C09134=1206.719,382.178,-78.740,-175.897,8.142,148.400
C09135=1206.716,382.425,-78.774,-175.896,8.145,148.400
C09136=1206.711,382.673,-78.809,-175.895,8.148,148.401
C09137=1206.707,382.920,-78.843,-175.894,8.151,148.401
C09138=1206.703,383.168,-78.877,-175.893,8.153,148.402
C09139=1206.700,383.415,-78.911,-175.892,8.156,148.402
C09140=1206.695,383.663,-78.946,-175.891,8.159,148.403
C09141=1206.691,383.911,-78.979,-175.890,8.162,148.403
C09142=1206.687,384.158,-79.014,-175.889,8.165,148.404
C09143=1206.684,384.406,-79.048,-175.888,8.168,148.404
C09144=1206.679,384.654,-79.082,-175.887,8.170,148.405
C09145=1206.675,384.901,-79.117,-175.887,8.173,148.405
C09146=1206.671,385.149,-79.151,-175.886,8.176,148.406
C09147=1206.667,385.396,-79.186,-175.885,8.179,148.406
C09148=1206.663,385.643,-79.219,-175.884,8.181,148.407
C09149=1206.659,385.892,-79.254,-175.883,8.185,148.407
C09150=1206.654,386.139,-79.289,-175.882,8.187,148.408
C09151=1206.651,386.387,-79.323,-175.882,8.190,148.408
C09152=1206.647,386.634,-79.357,-175.881,8.193,148.409
C09153=1206.643,386.881,-79.391,-175.880,8.196,148.409
C09154=1206.639,387.129,-79.426,-175.879,8.198,148.410
C09155=1206.634,387.377,-79.461,-175.878,8.201,148.410
C09156=1206.631,387.625,-79.495,-175.877,8.204,148.411
C09157=1206.626,387.872,-79.529,-175.876,8.207,148.411
C09158=1206.623,388.119,-79.563,-175.876,8.209,148.412
C09159=1206.619,388.367,-79.598,-175.875,8.212,148.412
C09160=1206.614,388.615,-79.633,-175.874,8.215,148.413
C09161=1206.611,388.863,-79.667,-175.874,8.217,148.413
C09162=1206.606,389.110,-79.701,-175.873,8.220,148.414
C09163=1206.602,389.358,-79.736,-175.872,8.223,148.414
C09164=1206.598,389.605,-79.770,-175.872,8.225,148.415
C09165=1206.594,389.853,-79.804,-175.870,8.228,148.415
C09166=1206.590,390.101,-79.839,-175.870,8.231,148.416
C09167=1206.586,390.348,-79.873,-175.869,8.233,148.416
C09168=1206.582,390.596,-79.908,-175.868,8.236,148.417
C09169=1206.577,390.843,-79.942,-175.867,8.239,148.417
C09170=1206.574,391.091,-79.977,-175.867,8.242,148.418
C09171=1206.570,391.338,-80.012,-175.866,8.244,148.418
C09172=1206.566,391.586,-80.047,-175.866,8.247,148.419
C09173=1206.562,391.833,-80.081,-175.865,8.250,148.419
C09174=1206.558,392.081,-80.115,-175.864,8.252,148.420
C09175=1206.553,392.364,-80.154,-175.864,8.255,148.420
C09176=1206.549,392.646,-80.194,-175.863,8.258,148.421
C09177=1206.544,392.928,-80.234,-175.862,8.261,148.421
C09178=1206.540,393.211,-80.273,-175.861,8.264,148.422
C09179=1206.535,393.459,-80.307,-175.861,8.267,148.423
C09180=1206.531,393.707,-80.342,-175.860,8.269,148.423
C09181=1206.527,393.954,-80.377,-175.859,8.272,148.423
C09182=1206.524,394.201,-80.412,-175.859,8.275,148.424
C09183=1206.519,394.449,-80.446,-175.858,8.277,148.424
C09184=1206.515,394.697,-80.481,-175.858,8.280,148.425
C09185=1206.511,394.944,-80.515,-175.857,8.283,148.425
C09186=1206.508,395.192,-80.550,-175.857,8.285,148.426
C09187=1206.503,395.439,-80.585,-175.856,8.287,148.426
C09188=1206.499,395.687,-80.620,-175.855,8.290,148.427
C09189=1206.495,395.935,-80.654,-175.855,8.292,148.427
C09190=1206.492,396.182,-80.689,-175.854,8.296,148.428
C09191=1206.487,396.429,-80.723,-175.853,8.297,148.428
C09192=1206.483,396.677,-80.758,-175.853,8.301,148.429
C09193=1206.479,396.925,-80.793,-175.853,8.303,148.430
C09194=1206.475,397.172,-80.828,-175.852,8.305,148.430
C09195=1206.471,397.419,-80.862,-175.851,8.308,148.430
C09196=1206.467,397.667,-80.897,-175.851,8.310,148.431
C09197=1206.463,397.915,-80.931,-175.851,8.312,148.432
C09198=1206.459,398.162,-80.967,-175.849,8.315,148.432
C09199=1206.454,398.410,-81.001,-175.849,8.318,148.432
C09200=1206.450,398.658,-81.036,-175.848,8.321,148.433
C09201=1206.447,398.904,-81.071,-175.848,8.323,148.434
C09202=1206.443,399.153,-81.106,-175.848,8.325,148.434
C09203=1206.438,399.400,-81.140,-175.847,8.328,148.435
C09204=1206.435,399.647,-81.176,-175.847,8.330,148.435
C09205=1206.430,399.895,-81.210,-175.846,8.333,148.436
C09206=1206.427,400.143,-81.244,-175.846,8.335,148.436
C09207=1206.423,400.389,-81.280,-175.845,8.338,148.437
C09208=1206.419,400.638,-81.314,-175.845,8.340,148.437
C09209=1206.414,400.885,-81.349,-175.845,8.342,148.438
C09210=1206.410,401.133,-81.384,-175.844,8.345,148.438
C09211=1206.406,401.380,-81.419,-175.843,8.347,148.439
C09212=1206.402,401.628,-81.454,-175.843,8.350,148.439
C09213=1206.399,401.875,-81.489,-175.843,8.352,148.440
C09214=1206.394,402.123,-81.523,-175.842,8.355,148.440
C09215=1206.391,402.370,-81.559,-175.841,8.357,148.441
C09216=1206.386,402.618,-81.593,-175.841,8.359,148.441
C09217=1206.382,402.866,-81.628,-175.841,8.361,148.442
C09218=1206.378,403.112,-81.663,-175.840,8.364,148.442
C09219=1206.374,403.361,-81.698,-175.839,8.366,148.443
C09220=1206.370,403.608,-81.734,-175.839,8.369,148.443
C09221=1206.366,403.856,-81.768,-175.839,8.371,148.444
C09222=1206.363,404.103,-81.802,-175.839,8.373,148.444
C09223=1206.358,404.350,-81.837,-175.838,8.376,148.445
C09224=1206.354,404.598,-81.872,-175.837,8.378,148.445
C09225=1206.350,404.845,-81.907,-175.837,8.381,148.446
C09226=1206.346,405.093,-81.942,-175.837,8.383,148.446
C09227=1206.342,405.341,-81.978,-175.837,8.385,148.447
C09228=1206.338,405.588,-82.012,-175.836,8.387,148.447
C09229=1206.334,405.836,-82.048,-175.836,8.389,148.447
C09230=1206.330,406.083,-82.082,-175.835,8.392,148.448
C09231=1206.326,406.331,-82.118,-175.835,8.395,148.449
C09232=1206.321,406.578,-82.152,-175.834,8.397,148.449
C09233=1206.318,406.825,-82.188,-175.834,8.399,148.449
C09234=1206.314,407.073,-82.222,-175.834,8.401,148.450
C09235=1206.310,407.320,-82.257,-175.833,8.404,148.451
C09236=1206.306,407.568,-82.292,-175.833,8.406,148.451
C09237=1206.302,407.815,-82.327,-175.833,8.408,148.451
C09238=1206.298,408.063,-82.362,-175.832,8.410,148.452
C09239=1206.294,408.311,-82.398,-175.832,8.413,148.453
C09240=1206.290,408.558,-82.432,-175.831,8.415,148.453
C09241=1206.286,408.806,-82.468,-175.831,8.417,148.453
C09242=1206.282,409.053,-82.502,-175.830,8.420,148.454
C09243=1206.278,409.300,-82.538,-175.830,8.422,148.454
C09244=1206.274,409.549,-82.573,-175.830,8.424,148.455
C09245=1206.270,409.795,-82.608,-175.829,8.426,148.455
C09246=1206.266,410.043,-82.643,-175.829,8.428,148.456
C09247=1206.262,410.291,-82.678,-175.829,8.431,148.456
C09248=1206.258,410.538,-82.713,-175.828,8.433,148.457
C09249=1206.254,410.786,-82.748,-175.828,8.435,148.457
C09250=1206.250,411.033,-82.783,-175.828,8.437,148.458
C09251=1206.246,411.281,-82.818,-175.828,8.439,148.458
C09252=1206.242,411.528,-82.854,-175.827,8.441,148.459
C09253=1206.238,411.775,-82.889,-175.827,8.444,148.459
C09254=1206.234,412.023,-82.924,-175.826,8.446,148.460
C09255=1206.230,412.271,-82.959,-175.826,8.448,148.460
C09256=1206.226,412.518,-82.994,-175.826,8.450,148.461
C09257=1206.222,412.766,-83.029,-175.825,8.452,148.461
C09258=1206.218,413.013,-83.065,-175.825,8.455,148.462
C09259=1206.214,413.261,-83.099,-175.824,8.457,148.462
C09260=1206.210,413.508,-83.135,-175.824,8.459,148.463
C09261=1206.206,413.755,-83.170,-175.824,8.461,148.463
C09262=1206.202,414.003,-83.205,-175.823,8.463,148.463
C09263=1206.198,414.250,-83.240,-175.823,8.465,148.464
C09264=1206.194,414.497,-83.276,-175.823,8.468,148.464
C09265=1206.190,414.745,-83.310,-175.822,8.470,148.465
C09266=1206.186,414.993,-83.346,-175.822,8.472,148.465
C09267=1206.182,415.240,-83.381,-175.822,8.474,148.466
C09268=1206.178,415.488,-83.416,-175.821,8.476,148.466
C09269=1206.174,415.735,-83.452,-175.821,8.478,148.467
C09270=1206.170,415.982,-83.487,-175.821,8.480,148.467
C09271=1206.165,416.261,-83.526,-175.820,8.483,148.468
C09272=1206.162,416.540,-83.566,-175.820,8.485,148.468
C09273=1206.160,416.817,-83.606,-175.820,8.487,148.469
C09274=1206.162,417.095,-83.644,-175.819,8.490,148.469
C09275=1205.741,417.096,-83.682,-175.823,8.500,148.473
C09276=1205.738,416.816,-83.643,-175.823,8.498,148.472
C09277=1205.740,416.534,-83.602,-175.823,8.496,148.472
C09278=1205.743,416.253,-83.563,-175.824,8.494,148.471
C09279=1205.748,415.972,-83.522,-175.825,8.491,148.471
C09280=1205.752,415.724,-83.488,-175.825,8.488,148.470
C09281=1205.756,415.477,-83.452,-175.824,8.487,148.470
C09282=1205.760,415.230,-83.417,-175.825,8.485,148.470
C09283=1205.764,414.981,-83.382,-175.825,8.483,148.469
C09284=1205.768,414.735,-83.347,-175.826,8.480,148.468
C09285=1205.772,414.487,-83.311,-175.826,8.478,148.468
C09286=1205.776,414.240,-83.277,-175.826,8.476,148.468
C09287=1205.780,413.992,-83.241,-175.827,8.474,148.467
C09288=1205.784,413.744,-83.205,-175.827,8.472,148.467
C09289=1205.789,413.497,-83.171,-175.828,8.470,148.466
C09290=1205.793,413.250,-83.135,-175.828,8.467,148.466
C09291=1205.796,413.002,-83.100,-175.828,8.465,148.465
C09292=1205.801,412.755,-83.065,-175.829,8.463,148.465
C09293=1205.804,412.507,-83.030,-175.829,8.461,148.464
C09294=1205.808,412.260,-82.994,-175.829,8.459,148.464
C09295=1205.813,412.012,-82.960,-175.829,8.456,148.463
C09296=1205.816,411.765,-82.924,-175.830,8.454,148.463
C09297=1205.820,411.517,-82.889,-175.830,8.452,148.462
C09298=1205.825,411.270,-82.854,-175.830,8.450,148.462
C09299=1205.828,411.022,-82.818,-175.831,8.448,148.461
C09300=1205.833,410.775,-82.784,-175.831,8.446,148.461
C09301=1205.836,410.527,-82.748,-175.832,8.443,148.460
C09302=1205.840,410.279,-82.714,-175.832,8.441,148.460
C09303=1205.845,410.032,-82.678,-175.832,8.439,148.459
C09304=1205.848,409.785,-82.643,-175.833,8.437,148.459
C09305=1205.852,409.537,-82.608,-175.833,8.435,148.459
C09306=1205.857,409.290,-82.573,-175.833,8.432,148.458
C09307=1205.861,409.042,-82.538,-175.833,8.430,148.457
C09308=1205.864,408.795,-82.503,-175.834,8.428,148.457
C09309=1205.868,408.547,-82.469,-175.834,8.426,148.457
C09310=1205.872,408.300,-82.433,-175.834,8.424,148.456
C09311=1205.876,408.052,-82.399,-175.835,8.421,148.456
C09312=1205.880,407.805,-82.363,-175.835,8.419,148.455
C09313=1205.884,407.558,-82.328,-175.836,8.416,148.455
C09314=1205.888,407.310,-82.293,-175.836,8.414,148.454
C09315=1205.892,407.062,-82.257,-175.836,8.412,148.454
C09316=1205.896,406.815,-82.223,-175.837,8.410,148.453
C09317=1205.900,406.568,-82.187,-175.837,8.407,148.453
C09318=1205.905,406.320,-82.153,-175.838,8.405,148.452
C09319=1205.908,406.073,-82.117,-175.838,8.403,148.452
C09320=1205.912,405.824,-82.083,-175.838,8.401,148.451
C09321=1205.916,405.578,-82.047,-175.839,8.398,148.451
C09322=1205.920,405.330,-82.013,-175.839,8.396,148.450
C09323=1205.925,405.082,-81.978,-175.840,8.393,148.450
C09324=1205.929,404.835,-81.943,-175.840,8.391,148.449
C09325=1205.932,404.587,-81.908,-175.841,8.389,148.449
C09326=1205.936,404.340,-81.873,-175.841,8.387,148.448
C09327=1205.940,404.092,-81.838,-175.841,8.384,148.448
C09328=1205.944,403.845,-81.803,-175.842,8.381,148.447
C09329=1205.948,403.597,-81.768,-175.842,8.379,148.447
C09330=1205.953,403.350,-81.733,-175.843,8.377,148.446
C09331=1205.957,403.102,-81.698,-175.843,8.375,148.446
C09332=1205.960,402.855,-81.663,-175.843,8.373,148.445
C09333=1205.965,402.607,-81.628,-175.844,8.369,148.445
C09334=1205.969,402.359,-81.593,-175.845,8.368,148.444
C09335=1205.972,402.113,-81.559,-175.845,8.365,148.444
C09336=1205.976,401.864,-81.524,-175.845,8.363,148.443
C09337=1205.981,401.618,-81.489,-175.846,8.360,148.443
C09338=1205.985,401.369,-81.454,-175.846,8.358,148.442
C09339=1205.989,401.122,-81.420,-175.847,8.356,148.442
C09340=1205.993,400.875,-81.384,-175.847,8.353,148.441
C09341=1205.997,400.626,-81.349,-175.848,8.350,148.441
C09342=1206.001,400.379,-81.315,-175.848,8.348,148.440
C09343=1206.004,400.132,-81.280,-175.848,8.346,148.440
C09344=1206.009,399.884,-81.245,-175.849,8.343,148.439
C09345=1206.013,399.636,-81.210,-175.849,8.341,148.439
C09346=1206.017,399.390,-81.175,-175.850,8.338,148.438
C09347=1206.021,399.141,-81.140,-175.851,8.336,148.438
C09348=1206.026,398.894,-81.106,-175.851,8.333,148.437
C09349=1206.029,398.647,-81.071,-175.851,8.331,148.437
C09350=1206.033,398.399,-81.037,-175.852,8.328,148.436
C09351=1206.037,398.151,-81.002,-175.853,8.326,148.436
C09352=1206.041,397.904,-80.967,-175.853,8.324,148.435
C09353=1206.045,397.656,-80.932,-175.854,8.321,148.435
C09354=1206.049,397.409,-80.898,-175.854,8.318,148.434
C09355=1206.053,397.162,-80.862,-175.855,8.316,148.434
C09356=1206.057,396.914,-80.828,-175.855,8.313,148.433
C09357=1206.061,396.666,-80.793,-175.856,8.311,148.433
C09358=1206.066,396.419,-80.758,-175.856,8.308,148.432
C09359=1206.069,396.172,-80.724,-175.857,8.306,148.432
C09360=1206.073,395.924,-80.689,-175.857,8.304,148.431
C09361=1206.077,395.676,-80.654,-175.858,8.301,148.430
C09362=1206.082,395.429,-80.620,-175.858,8.298,148.430
C09363=1206.086,395.181,-80.584,-175.859,8.295,148.430
C09364=1206.089,394.934,-80.550,-175.860,8.293,148.429
C09365=1206.093,394.686,-80.516,-175.860,8.290,148.428
C09366=1206.098,394.438,-80.481,-175.861,8.288,148.428
C09367=1206.102,394.190,-80.446,-175.862,8.285,148.428
C09368=1206.105,393.944,-80.412,-175.862,8.283,148.427
C09369=1206.109,393.696,-80.377,-175.863,8.280,148.426
C09370=1206.114,393.448,-80.342,-175.863,8.278,148.426
C09371=1206.118,393.200,-80.308,-175.864,8.275,148.425
C09372=1206.122,392.918,-80.268,-175.865,8.271,148.425
C09373=1206.127,392.635,-80.229,-175.865,8.269,148.424
C09374=1206.132,392.353,-80.189,-175.866,8.266,148.424
C09375=1206.136,392.070,-80.150,-175.867,8.263,148.423
C09376=1206.140,391.823,-80.114,-175.868,8.260,148.423
C09377=1206.144,391.576,-80.081,-175.868,8.258,148.422
C09378=1206.148,391.327,-80.046,-175.869,8.255,148.422
C09379=1206.152,391.080,-80.011,-175.870,8.252,148.421
C09380=1206.156,390.833,-79.977,-175.870,8.250,148.421
C09381=1206.160,390.585,-79.943,-175.871,8.247,148.420
C09382=1206.165,390.337,-79.908,-175.871,8.244,148.420
C09383=1206.168,390.090,-79.874,-175.873,8.241,148.419
C09384=1206.172,389.842,-79.839,-175.873,8.238,148.419
C09385=1206.176,389.595,-79.804,-175.874,8.236,148.418
C09386=1206.180,389.348,-79.770,-175.875,8.233,148.418
C09387=1206.184,389.099,-79.735,-175.876,8.230,148.417
C09388=1206.189,388.852,-79.701,-175.876,8.228,148.417
C09389=1206.192,388.605,-79.667,-175.877,8.225,148.416
C09390=1206.196,388.357,-79.632,-175.878,8.222,148.416
C09391=1206.201,388.109,-79.598,-175.878,8.220,148.415
C09392=1206.204,387.862,-79.563,-175.879,8.217,148.415
C09393=1206.209,387.614,-79.529,-175.880,8.214,148.414
C09394=1206.213,387.366,-79.494,-175.881,8.211,148.414
C09395=1206.217,387.119,-79.460,-175.881,8.209,148.413
C09396=1206.221,386.872,-79.426,-175.883,8.206,148.413
C09397=1206.225,386.623,-79.391,-175.883,8.203,148.412
C09398=1206.229,386.376,-79.357,-175.884,8.200,148.412
C09399=1206.233,386.128,-79.322,-175.885,8.198,148.411
C09400=1206.237,385.881,-79.288,-175.885,8.195,148.411
C09401=1206.241,385.634,-79.254,-175.887,8.192,148.410
C09402=1206.245,385.386,-79.219,-175.887,8.189,148.410
C09403=1206.249,385.138,-79.185,-175.888,8.187,148.409
C09404=1206.253,384.890,-79.150,-175.889,8.184,148.409
C09405=1206.257,384.643,-79.116,-175.890,8.181,148.408
C09406=1206.262,384.395,-79.083,-175.891,8.178,148.408
C09407=1206.265,384.147,-79.048,-175.892,8.175,148.407
C09408=1206.270,383.900,-79.014,-175.893,8.172,148.407
C09409=1206.274,383.652,-78.979,-175.894,8.169,148.406
C09410=1206.277,383.405,-78.945,-175.894,8.167,148.406
C09411=1206.282,383.157,-78.911,-175.895,8.164,148.405
C09412=1206.285,382.909,-78.877,-175.896,8.161,148.405
C09413=1206.290,382.662,-78.842,-175.897,8.158,148.404
C09414=1206.294,382.415,-78.808,-175.899,8.155,148.404
C09415=1206.298,382.166,-78.774,-175.899,8.152,148.403
C09416=1206.302,381.919,-78.740,-175.901,8.149,148.403
C09417=1206.306,381.672,-78.706,-175.901,8.146,148.402
C09418=1206.309,381.424,-78.671,-175.903,8.143,148.402
C09419=1206.314,381.176,-78.637,-175.904,8.141,148.402
C09420=1206.318,380.929,-78.604,-175.905,8.137,148.401
C09421=1206.322,380.681,-78.569,-175.906,8.135,148.401
C09422=1206.326,380.433,-78.535,-175.906,8.132,148.400
C09423=1206.331,380.186,-78.501,-175.907,8.130,148.400
C09424=1206.334,379.938,-78.466,-175.908,8.127,148.399
C09425=1206.339,379.690,-78.433,-175.909,8.124,148.399
C09426=1206.342,379.443,-78.399,-175.910,8.121,148.398
C09427=1206.346,379.195,-78.364,-175.912,8.118,148.398
C09428=1206.350,378.948,-78.330,-175.912,8.115,148.397
C09429=1206.355,378.700,-78.296,-175.914,8.111,148.397
C09430=1206.359,378.453,-78.263,-175.915,8.108,148.397
C09431=1206.363,378.205,-78.228,-175.916,8.105,148.396
C09432=1206.367,377.957,-78.195,-175.917,8.103,148.396
C09433=1206.371,377.710,-78.161,-175.918,8.100,148.395
C09434=1206.375,377.462,-78.126,-175.920,8.097,148.395
C09435=1206.379,377.215,-78.092,-175.920,8.094,148.394
C09436=1206.384,376.966,-78.058,-175.922,8.091,148.394
C09437=1206.387,376.719,-78.024,-175.923,8.088,148.393
C09438=1206.392,376.471,-77.990,-175.924,8.085,148.393
C09439=1206.396,376.224,-77.956,-175.925,8.083,148.393
C09440=1206.399,375.976,-77.922,-175.926,8.079,148.392
C09441=1206.404,375.728,-77.888,-175.927,8.077,148.392
C09442=1206.407,375.481,-77.854,-175.929,8.073,148.391
C09443=1206.411,375.233,-77.821,-175.930,8.070,148.391
C09444=1206.416,374.985,-77.787,-175.931,8.067,148.390
C09445=1206.419,374.738,-77.753,-175.933,8.065,148.390
C09446=1206.424,374.490,-77.719,-175.933,8.062,148.389
C09447=1206.428,374.242,-77.685,-175.935,8.059,148.389
C09448=1206.432,373.995,-77.652,-175.936,8.055,148.389
C09449=1206.436,373.747,-77.617,-175.938,8.052,148.388
C09450=1206.440,373.500,-77.583,-175.939,8.049,148.388
C09451=1206.444,373.252,-77.550,-175.940,8.047,148.387
C09452=1206.449,373.004,-77.516,-175.941,8.044,148.387
C09453=1206.452,372.756,-77.482,-175.943,8.040,148.387
C09454=1206.456,372.509,-77.448,-175.944,8.037,148.386
C09455=1206.461,372.261,-77.414,-175.945,8.035,148.386
C09456=1206.465,372.014,-77.381,-175.947,8.032,148.385
C09457=1206.468,371.765,-77.347,-175.948,8.029,148.385
C09458=1206.472,371.518,-77.313,-175.950,8.025,148.385
C09459=1206.477,371.270,-77.279,-175.951,8.022,148.384
C09460=1206.481,371.022,-77.246,-175.952,8.020,148.384
C09461=1206.485,370.775,-77.212,-175.953,8.017,148.383
C09462=1206.489,370.527,-77.179,-175.955,8.013,148.383
C09463=1206.493,370.279,-77.144,-175.956,8.010,148.383
C09464=1206.497,370.032,-77.111,-175.957,8.008,148.382
C09465=1206.501,369.784,-77.078,-175.959,8.004,148.382
C09466=1206.505,369.537,-77.044,-175.960,8.001,148.381
C09467=1206.510,369.288,-77.010,-175.961,7.998,148.381
C09468=1206.513,369.041,-76.976,-175.963,7.996,148.381
C09469=1206.517,368.793,-76.943,-175.964,7.992,148.380
C09470=1206.522,368.546,-76.910,-175.966,7.989,148.380
C09471=1206.526,368.298,-76.875,-175.967,7.987,148.380
C09472=1206.530,368.050,-76.842,-175.969,7.983,148.379
C09473=1206.534,367.802,-76.809,-175.970,7.980,148.379
C09474=1206.538,367.555,-76.775,-175.971,7.977,148.378
C09475=1206.542,367.307,-76.742,-175.973,7.974,148.378
C09476=1206.547,367.026,-76.703,-175.975,7.970,148.377
C09477=1206.551,366.746,-76.666,-175.977,7.967,148.377
C09478=1206.556,366.466,-76.628,-175.978,7.964,148.377
C09479=1206.560,366.185,-76.590,-175.980,7.960,148.376
C09480=1206.565,365.937,-76.556,-175.981,7.957,148.376
C09481=1206.569,365.690,-76.523,-175.983,7.954,148.376
C09482=1206.573,365.442,-76.490,-175.985,7.951,148.375
C09483=1206.577,365.195,-76.456,-175.987,7.948,148.375
C09484=1206.581,364.947,-76.423,-175.988,7.945,148.375
C09485=1206.585,364.699,-76.389,-175.989,7.942,148.374
C09486=1206.589,364.451,-76.356,-175.991,7.939,148.374
C09487=1206.593,364.203,-76.323,-175.992,7.936,148.374
C09488=1206.597,363.956,-76.289,-175.994,7.932,148.373
C09489=1206.601,363.708,-76.256,-175.996,7.930,148.373
C09490=1206.605,363.461,-76.223,-175.998,7.926,148.372
C09491=1206.610,363.213,-76.189,-175.999,7.924,148.372
C09492=1206.614,362.965,-76.156,-176.000,7.921,148.372
C09493=1206.618,362.717,-76.123,-176.002,7.917,148.371
C09494=1206.623,362.469,-76.090,-176.004,7.915,148.371
C09495=1206.627,362.222,-76.057,-176.006,7.911,148.371
C09496=1206.630,361.973,-76.023,-176.007,7.908,148.371
C09497=1206.634,361.726,-75.989,-176.009,7.905,148.370
C09498=1206.638,361.478,-75.956,-176.010,7.902,148.370
C09499=1206.642,361.231,-75.923,-176.012,7.899,148.370
C09500=1206.646,360.983,-75.890,-176.014,7.896,148.369
C09501=1206.651,360.735,-75.857,-176.016,7.892,148.369
C09502=1206.655,360.487,-75.823,-176.017,7.890,148.369
C09503=1206.659,360.240,-75.790,-176.019,7.886,148.368
C09504=1206.663,359.992,-75.757,-176.020,7.883,148.368
C09505=1206.667,359.744,-75.724,-176.023,7.880,148.368
C09506=1206.671,359.497,-75.691,-176.024,7.877,148.367
C09507=1206.675,359.249,-75.658,-176.026,7.874,148.367
C09508=1206.680,359.000,-75.625,-176.028,7.871,148.367
C09509=1206.684,358.753,-75.592,-176.030,7.868,148.366
C09510=1206.688,358.505,-75.559,-176.031,7.865,148.366
C09511=1206.692,358.258,-75.526,-176.033,7.862,148.366
C09512=1206.696,358.010,-75.493,-176.035,7.859,148.366
C09513=1206.700,357.762,-75.460,-176.036,7.855,148.365
C09514=1206.704,357.514,-75.427,-176.038,7.853,148.365
C09515=1206.708,357.267,-75.394,-176.040,7.850,148.365
C09516=1206.712,357.019,-75.360,-176.041,7.847,148.364
C09517=1206.717,356.771,-75.328,-176.044,7.843,148.364
C09518=1206.721,356.523,-75.295,-176.045,7.841,148.364
C09519=1206.725,356.275,-75.262,-176.047,7.837,148.364
C09520=1206.729,356.027,-75.229,-176.049,7.835,148.363
C09521=1206.733,355.780,-75.196,-176.051,7.831,148.363
C09522=1206.737,355.532,-75.164,-176.053,7.828,148.363
C09523=1206.741,355.284,-75.130,-176.054,7.825,148.363
C09524=1206.745,355.036,-75.097,-176.057,7.822,148.362
C09525=1206.749,354.788,-75.064,-176.058,7.819,148.362
C09526=1206.754,354.540,-75.032,-176.060,7.816,148.362
C09527=1206.757,354.293,-74.999,-176.062,7.813,148.362
C09528=1206.761,354.045,-74.966,-176.064,7.810,148.361
C09529=1206.765,353.797,-74.933,-176.065,7.807,148.361
C09530=1206.770,353.549,-74.900,-176.067,7.804,148.361
C09531=1206.775,353.302,-74.868,-176.069,7.801,148.360
C09532=1206.778,353.054,-74.835,-176.071,7.798,148.360
C09533=1206.783,352.806,-74.803,-176.073,7.795,148.360
C09534=1206.787,352.558,-74.769,-176.075,7.792,148.360
C09535=1206.791,352.311,-74.736,-176.077,7.788,148.359
C09536=1206.795,352.062,-74.704,-176.078,7.786,148.359
C09537=1206.799,351.815,-74.671,-176.081,7.783,148.359
C09538=1206.803,351.566,-74.639,-176.082,7.780,148.359
C09539=1206.807,351.319,-74.606,-176.084,7.776,148.358
C09540=1206.811,351.071,-74.572,-176.086,7.774,148.358
C09541=1206.816,350.824,-74.541,-176.088,7.771,148.358
C09542=1206.820,350.576,-74.508,-176.090,7.767,148.358
C09543=1206.824,350.328,-74.475,-176.092,7.765,148.358
C09544=1206.828,350.080,-74.443,-176.094,7.761,148.357
C09545=1206.832,349.832,-74.410,-176.096,7.759,148.357
C09546=1206.836,349.584,-74.377,-176.098,7.756,148.357
C09547=1206.841,349.336,-74.345,-176.099,7.753,148.357
C09548=1206.845,349.089,-74.313,-176.101,7.749,148.356
C09549=1206.849,348.841,-74.280,-176.103,7.746,148.356
C09550=1206.853,348.593,-74.247,-176.105,7.744,148.356
C09551=1206.857,348.345,-74.215,-176.107,7.740,148.356
C09552=1206.861,348.097,-74.182,-176.109,7.738,148.356
C09553=1206.865,347.849,-74.150,-176.111,7.734,148.355
C09554=1206.870,347.602,-74.117,-176.113,7.731,148.355
C09555=1206.874,347.354,-74.085,-176.115,7.728,148.355
C09556=1206.878,347.106,-74.053,-176.117,7.725,148.355
C09557=1206.882,346.858,-74.020,-176.119,7.723,148.355
C09558=1206.886,346.610,-73.988,-176.121,7.719,148.354
C09559=1206.891,346.362,-73.956,-176.123,7.717,148.354
C09560=1206.895,346.115,-73.923,-176.125,7.713,148.354
C09561=1206.898,345.867,-73.891,-176.127,7.710,148.354
C09562=1206.903,345.619,-73.858,-176.129,7.708,148.353
C09563=1206.907,345.370,-73.825,-176.131,7.704,148.353
C09564=1206.911,345.123,-73.794,-176.133,7.702,148.353
C09565=1206.916,344.875,-73.762,-176.135,7.698,148.353
C09566=1206.919,344.627,-73.729,-176.137,7.695,148.353
C09567=1206.924,344.379,-73.697,-176.139,7.692,148.352
C09568=1206.928,344.132,-73.665,-176.141,7.689,148.352
C09569=1206.932,343.883,-73.633,-176.143,7.687,148.352
C09570=1206.936,343.636,-73.600,-176.145,7.683,148.352
C09571=1206.940,343.388,-73.568,-176.147,7.681,148.352
C09572=1206.945,343.140,-73.536,-176.149,7.678,148.352
C09573=1206.949,342.892,-73.504,-176.152,7.674,148.351
C09574=1206.952,342.644,-73.471,-176.153,7.672,148.351
C09575=1206.957,342.396,-73.439,-176.155,7.669,148.351
C09576=1206.961,342.149,-73.407,-176.157,7.666,148.351
C09577=1206.966,341.900,-73.375,-176.159,7.663,148.351
C09578=1206.969,341.652,-73.343,-176.161,7.659,148.350
C09579=1206.974,341.404,-73.310,-176.164,7.657,148.350
C09580=1206.978,341.126,-73.275,-176.166,7.654,148.350
C09581=1206.983,340.849,-73.239,-176.168,7.650,148.350
C09582=1206.988,340.570,-73.202,-176.170,7.647,148.350
C09583=1206.993,340.292,-73.167,-176.172,7.644,148.350
C09584=1206.997,340.044,-73.135,-176.175,7.640,148.349
C09585=1207.001,339.796,-73.103,-176.177,7.637,148.349
C09586=1207.005,339.548,-73.071,-176.179,7.635,148.349
C09587=1207.009,339.300,-73.039,-176.181,7.632,148.349
C09588=1207.014,339.052,-73.007,-176.183,7.629,148.349
C09589=1207.018,338.804,-72.975,-176.186,7.626,148.349
C09590=1207.022,338.556,-72.943,-176.188,7.623,148.348
C09591=1207.027,338.308,-72.911,-176.189,7.620,148.348
C09592=1207.030,338.060,-72.879,-176.192,7.617,148.348
C09593=1207.034,337.812,-72.847,-176.194,7.615,148.348
C09594=1207.039,337.565,-72.815,-176.196,7.611,148.348
C09595=1207.043,337.317,-72.784,-176.198,7.608,148.348
C09596=1207.046,337.069,-72.752,-176.200,7.605,148.348
C09597=1207.051,336.821,-72.720,-176.202,7.602,148.348
C09598=1207.055,336.573,-72.688,-176.205,7.599,148.347
C09599=1207.059,336.325,-72.656,-176.206,7.596,148.347
C09600=1207.063,336.078,-72.624,-176.209,7.593,148.347
C09601=1207.068,335.829,-72.592,-176.211,7.591,148.347
C09602=1207.071,335.581,-72.560,-176.213,7.588,148.347
C09603=1207.076,335.333,-72.529,-176.215,7.584,148.346
C09604=1207.080,335.085,-72.498,-176.217,7.582,148.347
C09605=1207.085,334.838,-72.465,-176.219,7.579,148.346
C09606=1207.088,334.590,-72.434,-176.221,7.576,148.346
C09607=1207.093,334.342,-72.402,-176.224,7.573,148.346
C09608=1207.097,334.094,-72.371,-176.226,7.570,148.346
C09609=1207.101,333.845,-72.339,-176.228,7.568,148.346
C09610=1207.106,333.598,-72.307,-176.230,7.564,148.346
C09611=1207.109,333.350,-72.275,-176.232,7.562,148.346
C09612=1207.114,333.102,-72.244,-176.235,7.559,148.346
C09613=1207.118,332.854,-72.213,-176.237,7.555,148.345
C09614=1207.123,332.606,-72.181,-176.239,7.553,148.345
C09615=1207.126,332.358,-72.149,-176.241,7.550,148.345
C09616=1207.130,332.109,-72.118,-176.243,7.546,148.345
C09617=1207.135,331.862,-72.086,-176.246,7.544,148.345
C09618=1207.138,331.614,-72.054,-176.248,7.541,148.345
C09619=1207.143,331.366,-72.024,-176.249,7.538,148.345
C09620=1207.147,331.118,-71.991,-176.252,7.535,148.345
C09621=1207.152,330.870,-71.960,-176.254,7.532,148.344
C09622=1207.156,330.622,-71.928,-176.256,7.530,148.344
C09623=1207.160,330.374,-71.897,-176.259,7.526,148.344
C09624=1207.164,330.126,-71.866,-176.261,7.524,148.344
C09625=1207.168,329.878,-71.834,-176.263,7.521,148.344
C09626=1207.172,329.630,-71.803,-176.266,7.518,148.344
C09627=1207.177,329.382,-71.772,-176.267,7.515,148.344
C09628=1207.180,329.134,-71.740,-176.270,7.512,148.344
C09629=1207.185,328.886,-71.709,-176.272,7.510,148.344
C09630=1207.189,328.638,-71.677,-176.274,7.507,148.343
C09631=1207.194,328.390,-71.646,-176.277,7.503,148.343
C09632=1207.198,328.142,-71.614,-176.278,7.501,148.343
C09633=1207.202,327.894,-71.583,-176.281,7.498,148.343
C09634=1207.206,327.646,-71.551,-176.284,7.495,148.343
C09635=1207.211,327.398,-71.521,-176.285,7.492,148.343
C09636=1207.214,327.150,-71.489,-176.288,7.489,148.343
C09637=1207.219,326.902,-71.458,-176.290,7.487,148.343
C09638=1207.223,326.654,-71.427,-176.292,7.484,148.343
C09639=1207.227,326.406,-71.396,-176.294,7.480,148.343
C09640=1207.232,326.158,-71.365,-176.297,7.478,148.343
C09641=1207.236,325.910,-71.333,-176.299,7.475,148.343
C09642=1207.240,325.662,-71.302,-176.301,7.473,148.343
C09643=1207.244,325.414,-71.271,-176.303,7.469,148.342
C09644=1207.249,325.166,-71.240,-176.306,7.466,148.342
C09645=1207.252,324.918,-71.209,-176.308,7.464,148.342
C09646=1207.256,324.670,-71.178,-176.310,7.461,148.342
C09647=1207.261,324.423,-71.147,-176.313,7.458,148.342
C09648=1207.265,324.174,-71.116,-176.314,7.455,148.342
C09649=1207.269,323.926,-71.085,-176.317,7.452,148.342
C09650=1207.273,323.678,-71.053,-176.319,7.450,148.342
C09651=1207.278,323.430,-71.022,-176.321,7.447,148.342
C09652=1207.282,323.182,-70.991,-176.324,7.444,148.342
C09653=1207.286,322.933,-70.960,-176.326,7.441,148.342
C09654=1207.290,322.686,-70.929,-176.328,7.438,148.342
C09655=1207.294,322.438,-70.898,-176.331,7.436,148.342
C09656=1207.298,322.190,-70.868,-176.333,7.433,148.342
C09657=1207.303,321.942,-70.837,-176.335,7.429,148.342
C09658=1207.307,321.693,-70.806,-176.337,7.427,148.341
C09659=1207.311,321.446,-70.774,-176.340,7.424,148.341
C09660=1207.316,321.198,-70.743,-176.342,7.422,148.341
C09661=1207.319,320.949,-70.713,-176.344,7.418,148.341
C09662=1207.324,320.701,-70.682,-176.347,7.415,148.341
C09663=1207.329,320.454,-70.651,-176.349,7.413,148.341
C09664=1207.333,320.205,-70.620,-176.351,7.410,148.341
C09665=1207.337,319.957,-70.589,-176.353,7.408,148.341
C09666=1207.341,319.709,-70.559,-176.356,7.405,148.341
C09667=1207.345,319.461,-70.527,-176.359,7.402,148.341
C09668=1207.349,319.213,-70.497,-176.360,7.399,148.341
C09669=1207.354,318.965,-70.466,-176.363,7.396,148.341
C09670=1207.357,318.717,-70.435,-176.366,7.393,148.341
C09671=1207.362,318.469,-70.405,-176.367,7.390,148.341
C09672=1207.366,318.221,-70.374,-176.370,7.387,148.341
C09673=1207.371,317.973,-70.343,-176.372,7.385,148.341
C09674=1207.374,317.725,-70.313,-176.374,7.382,148.341
C09675=1207.379,317.477,-70.282,-176.377,7.379,148.341
C09676=1207.384,317.229,-70.251,-176.379,7.377,148.341
C09677=1207.387,316.980,-70.221,-176.382,7.374,148.341
C09678=1207.391,316.733,-70.190,-176.383,7.371,148.341
C09679=1207.396,316.485,-70.159,-176.386,7.368,148.341
C09680=1207.400,316.236,-70.130,-176.389,7.365,148.341
C09681=1207.404,315.988,-70.098,-176.391,7.363,148.341
C09682=1207.409,315.740,-70.068,-176.393,7.359,148.340
C09683=1207.413,315.492,-70.037,-176.395,7.357,148.340
C09684=1207.418,315.216,-70.003,-176.398,7.354,148.340
C09685=1207.423,314.940,-69.970,-176.401,7.351,148.340
C09686=1207.427,314.663,-69.935,-176.403,7.348,148.340
C09687=1207.432,314.387,-69.901,-176.406,7.345,148.340
C09688=1207.436,314.139,-69.871,-176.409,7.342,148.340
C09689=1207.440,313.891,-69.840,-176.411,7.339,148.340
C09690=1207.445,313.643,-69.810,-176.413,7.337,148.340
C09691=1207.448,313.395,-69.779,-176.416,7.334,148.340
C09692=1207.453,313.146,-69.749,-176.418,7.331,148.340
C09693=1207.457,312.899,-69.719,-176.420,7.328,148.340
C09694=1207.462,312.651,-69.688,-176.422,7.326,148.340
C09695=1207.466,312.403,-69.658,-176.425,7.323,148.340
C09696=1207.470,312.155,-69.628,-176.428,7.320,148.340
C09697=1207.474,311.906,-69.597,-176.430,7.318,148.340
C09698=1207.478,311.658,-69.567,-176.432,7.315,148.340
C09699=1207.483,311.410,-69.537,-176.434,7.312,148.340
C09700=1207.487,311.162,-69.506,-176.437,7.309,148.340
C09701=1207.492,310.914,-69.476,-176.439,7.306,148.340
C09702=1207.496,310.666,-69.446,-176.441,7.304,148.340
C09703=1207.500,310.417,-69.415,-176.444,7.301,148.340
C09704=1207.504,310.170,-69.385,-176.446,7.299,148.340
C09705=1207.509,309.921,-69.355,-176.449,7.295,148.340
C09706=1207.513,309.673,-69.325,-176.451,7.293,148.340
C09707=1207.518,309.425,-69.295,-176.453,7.290,148.340
C09708=1207.521,309.177,-69.265,-176.456,7.287,148.340
C09709=1207.525,308.929,-69.234,-176.458,7.285,148.340
C09710=1207.530,308.681,-69.204,-176.461,7.282,148.340
C09711=1207.534,308.433,-69.174,-176.463,7.279,148.340
C09712=1207.538,308.184,-69.144,-176.466,7.276,148.340
C09713=1207.542,307.936,-69.114,-176.468,7.273,148.340
C09714=1207.547,307.688,-69.084,-176.470,7.271,148.340
C09715=1207.551,307.440,-69.053,-176.473,7.268,148.340
C09716=1207.555,307.192,-69.024,-176.475,7.266,148.340
C09717=1207.560,306.944,-68.993,-176.478,7.263,148.340
C09718=1207.564,306.696,-68.964,-176.480,7.260,148.340
C09719=1207.569,306.447,-68.934,-176.482,7.257,148.340
C09720=1207.573,306.199,-68.903,-176.485,7.254,148.340
C09721=1207.577,305.951,-68.874,-176.487,7.252,148.340
C09722=1207.582,305.703,-68.843,-176.490,7.249,148.340
C09723=1207.586,305.455,-68.814,-176.492,7.247,148.340
C09724=1207.590,305.207,-68.784,-176.495,7.244,148.340
C09725=1207.595,304.959,-68.754,-176.497,7.242,148.340
C09726=1207.599,304.710,-68.724,-176.499,7.239,148.340
C09727=1207.603,304.463,-68.694,-176.501,7.237,148.340
C09728=1207.606,304.214,-68.664,-176.504,7.233,148.341
C09729=1207.611,303.965,-68.634,-176.507,7.230,148.341
C09730=1207.615,303.717,-68.605,-176.509,7.228,148.341
C09731=1207.619,303.469,-68.574,-176.512,7.225,148.341
C09732=1207.624,303.221,-68.544,-176.514,7.223,148.341
C09733=1207.628,302.972,-68.515,-176.516,7.220,148.341
C09734=1207.632,302.725,-68.485,-176.519,7.218,148.341
C09735=1207.636,302.476,-68.455,-176.521,7.215,148.341
C09736=1207.641,302.228,-68.425,-176.523,7.213,148.341
C09737=1207.646,301.980,-68.396,-176.526,7.210,148.341
C09738=1207.650,301.732,-68.367,-176.529,7.207,148.341
C09739=1207.654,301.484,-68.337,-176.531,7.204,148.341
C09740=1207.658,301.236,-68.307,-176.534,7.201,148.341
C09741=1207.663,300.988,-68.277,-176.536,7.199,148.341
C09742=1207.667,300.739,-68.248,-176.538,7.196,148.341
C09743=1207.672,300.491,-68.218,-176.541,7.194,148.341
C09744=1207.676,300.243,-68.189,-176.543,7.191,148.341
C09745=1207.680,299.995,-68.159,-176.545,7.189,148.341
C09746=1207.684,299.747,-68.129,-176.548,7.186,148.341
C09747=1207.689,299.498,-68.099,-176.550,7.183,148.341
C09748=1207.693,299.250,-68.070,-176.553,7.180,148.341
C09749=1207.697,299.002,-68.040,-176.556,7.177,148.341
C09750=1207.701,298.753,-68.011,-176.558,7.175,148.341
C09751=1207.706,298.505,-67.981,-176.560,7.172,148.341
C09752=1207.710,298.257,-67.952,-176.562,7.170,148.341
C09753=1207.714,298.009,-67.922,-176.565,7.167,148.341
C09754=1207.718,297.760,-67.893,-176.567,7.165,148.341
C09755=1207.724,297.513,-67.863,-176.570,7.162,148.341
C09756=1207.728,297.264,-67.834,-176.573,7.160,148.342
C09757=1207.732,297.016,-67.804,-176.575,7.157,148.342
C09758=1207.736,296.768,-67.775,-176.577,7.155,148.342
C09759=1207.740,296.519,-67.745,-176.580,7.152,148.342
C09760=1207.744,296.271,-67.716,-176.582,7.149,148.342
C09761=1207.749,296.023,-67.686,-176.585,7.146,148.342
C09762=1207.753,295.775,-67.657,-176.587,7.144,148.342
C09763=1207.758,295.527,-67.628,-176.590,7.141,148.342
C09764=1207.762,295.279,-67.598,-176.592,7.139,148.342
C09765=1207.766,295.030,-67.570,-176.595,7.136,148.342
C09766=1207.770,294.782,-67.540,-176.597,7.133,148.342
C09767=1207.775,294.533,-67.511,-176.600,7.131,148.342
C09768=1207.779,294.285,-67.481,-176.602,7.128,148.342
C09769=1207.783,294.037,-67.452,-176.605,7.126,148.342
C09770=1207.788,293.789,-67.423,-176.607,7.123,148.342
C09771=1207.792,293.540,-67.394,-176.609,7.121,148.343
C09772=1207.796,293.292,-67.365,-176.612,7.117,148.343
C09773=1207.801,293.044,-67.335,-176.614,7.115,148.343
C09774=1207.804,292.796,-67.306,-176.617,7.112,148.343
C09775=1207.809,292.548,-67.277,-176.620,7.110,148.343
C09776=1207.813,292.299,-67.249,-176.622,7.107,148.343
C09777=1207.818,292.051,-67.219,-176.624,7.105,148.343
C09778=1207.822,291.803,-67.190,-176.627,7.102,148.343
C09779=1207.826,291.555,-67.160,-176.629,7.100,148.343
C09780=1207.831,291.307,-67.132,-176.632,7.097,148.343
C09781=1207.835,291.058,-67.102,-176.634,7.095,148.343
C09782=1207.839,290.810,-67.073,-176.637,7.092,148.343
C09783=1207.843,290.561,-67.045,-176.639,7.090,148.343
C09784=1207.847,290.313,-67.015,-176.642,7.087,148.344
C09785=1207.852,290.066,-66.986,-176.644,7.085,148.344
C09786=1207.857,289.817,-66.957,-176.647,7.082,148.344
C09787=1207.861,289.568,-66.928,-176.649,7.079,148.344
C09788=1207.866,289.294,-66.896,-176.652,7.077,148.344
C09789=1207.870,289.020,-66.865,-176.655,7.074,148.344
C09790=1207.875,288.746,-66.832,-176.657,7.071,148.344
C09791=1207.880,288.472,-66.801,-176.660,7.069,148.344
C09792=1207.884,288.223,-66.772,-176.663,7.066,148.344
C09793=1207.888,287.974,-66.743,-176.665,7.064,148.344
C09794=1207.893,287.727,-66.713,-176.668,7.061,148.344
C09795=1207.898,287.478,-66.685,-176.670,7.058,148.344
C09796=1207.901,287.230,-66.656,-176.673,7.056,148.345
C09797=1207.906,286.982,-66.627,-176.675,7.053,148.345
C09798=1207.910,286.734,-66.598,-176.678,7.050,148.345
C09799=1207.915,286.485,-66.569,-176.680,7.048,148.345
C09800=1207.919,286.237,-66.542,-176.683,7.045,148.345
C09801=1207.923,285.989,-66.512,-176.685,7.043,148.345
C09802=1207.928,285.740,-66.483,-176.688,7.040,148.345
C09803=1207.932,285.492,-66.455,-176.690,7.038,148.345
C09804=1207.936,285.243,-66.426,-176.693,7.035,148.345
C09805=1207.941,284.995,-66.397,-176.695,7.033,148.346
C09806=1207.945,284.747,-66.369,-176.698,7.030,148.346
C09807=1207.949,284.498,-66.340,-176.700,7.028,148.346
C09808=1207.954,284.250,-66.311,-176.702,7.026,148.346
C09809=1207.958,284.002,-66.283,-176.705,7.023,148.346
C09810=1207.962,283.753,-66.254,-176.707,7.021,148.346
C09811=1207.967,283.505,-66.225,-176.710,7.018,148.346
C09812=1207.971,283.257,-66.197,-176.712,7.016,148.346
C09813=1207.975,283.008,-66.168,-176.715,7.013,148.346
C09814=1207.981,282.760,-66.140,-176.718,7.011,148.346
C09815=1207.984,282.512,-66.111,-176.720,7.008,148.346
C09816=1207.988,282.263,-66.082,-176.722,7.006,148.347
C09817=1207.993,282.016,-66.054,-176.726,7.003,148.347
C09818=1207.997,281.767,-66.026,-176.728,7.001,148.347
C09819=1208.002,281.519,-65.997,-176.730,6.998,148.347
C09820=1208.006,281.270,-65.968,-176.733,6.995,148.347
C09821=1208.010,281.022,-65.940,-176.735,6.994,148.347
C09822=1208.015,280.774,-65.912,-176.738,6.991,148.347
C09823=1208.019,280.525,-65.883,-176.740,6.988,148.347
C09824=1208.023,280.278,-65.855,-176.743,6.986,148.348
C09825=1208.028,280.029,-65.826,-176.745,6.983,148.348
C09826=1208.031,279.780,-65.798,-176.747,6.981,148.348
C09827=1208.037,279.532,-65.769,-176.750,6.978,148.348
C09828=1208.040,279.283,-65.741,-176.753,6.976,148.348
C09829=1208.045,279.035,-65.713,-176.755,6.973,148.348
C09830=1208.049,278.787,-65.685,-176.758,6.971,148.348
C09831=1208.054,278.538,-65.656,-176.761,6.968,148.348
C09832=1208.058,278.290,-65.628,-176.763,6.966,148.348
C09833=1208.063,278.042,-65.599,-176.765,6.964,148.349
C09834=1208.066,277.794,-65.571,-176.768,6.961,148.349
C09835=1208.072,277.545,-65.543,-176.770,6.959,148.349
C09836=1208.075,277.297,-65.515,-176.773,6.956,148.349
C09837=1208.080,277.049,-65.486,-176.776,6.954,148.349
C09838=1208.084,276.800,-65.458,-176.778,6.951,148.349
C09839=1208.088,276.552,-65.430,-176.780,6.949,148.349
C09840=1208.093,276.303,-65.402,-176.783,6.947,148.350
C09841=1208.097,276.056,-65.374,-176.786,6.944,148.350
C09842=1208.102,275.806,-65.346,-176.788,6.942,148.350
C09843=1208.106,275.558,-65.318,-176.791,6.939,148.350
C09844=1208.110,275.310,-65.290,-176.793,6.937,148.350
C09845=1208.115,275.061,-65.261,-176.795,6.935,148.350
C09846=1208.119,274.813,-65.233,-176.798,6.932,148.350
C09847=1208.123,274.565,-65.206,-176.801,6.930,148.350
C09848=1208.128,274.316,-65.177,-176.803,6.927,148.350
C09849=1208.132,274.068,-65.149,-176.806,6.925,148.351
C09850=1208.136,273.820,-65.121,-176.808,6.923,148.351
C09851=1208.141,273.571,-65.093,-176.811,6.920,148.351
C09852=1208.145,273.322,-65.065,-176.813,6.918,148.351
C09853=1208.149,273.074,-65.037,-176.816,6.915,148.351
C09854=1208.155,272.826,-65.009,-176.818,6.913,148.351
C09855=1208.158,272.578,-64.981,-176.821,6.911,148.352
C09856=1208.163,272.329,-64.954,-176.823,6.908,148.352
C09857=1208.167,272.080,-64.925,-176.826,6.906,148.352
C09858=1208.172,271.832,-64.897,-176.828,6.904,148.352
C09859=1208.176,271.584,-64.869,-176.831,6.901,148.352
C09860=1208.180,271.335,-64.842,-176.834,6.899,148.352
C09861=1208.185,271.087,-64.814,-176.836,6.896,148.352
C09862=1208.189,270.838,-64.785,-176.839,6.894,148.353
C09863=1208.193,270.591,-64.758,-176.841,6.892,148.353
C09864=1208.198,270.342,-64.731,-176.844,6.889,148.353
C09865=1208.203,270.093,-64.702,-176.846,6.887,148.353
C09866=1208.207,269.845,-64.674,-176.848,6.885,148.353
C09867=1208.211,269.596,-64.647,-176.852,6.882,148.353
C09868=1208.215,269.348,-64.619,-176.854,6.880,148.353
C09869=1208.220,269.100,-64.591,-176.856,6.877,148.354
C09870=1208.224,268.851,-64.563,-176.859,6.875,148.354
C09871=1208.229,268.603,-64.535,-176.861,6.873,148.354
C09872=1208.233,268.354,-64.508,-176.864,6.870,148.354
C09873=1208.237,268.106,-64.480,-176.866,6.868,148.354
C09874=1208.242,267.857,-64.453,-176.869,6.866,148.354
C09875=1208.246,267.610,-64.425,-176.872,6.863,148.355
C09876=1208.250,267.361,-64.397,-176.874,6.861,148.355
C09877=1208.255,267.112,-64.369,-176.877,6.859,148.355
C09878=1208.260,266.864,-64.342,-176.879,6.856,148.355
C09879=1208.264,266.615,-64.314,-176.882,6.854,148.355
C09880=1208.268,266.367,-64.287,-176.884,6.852,148.355
C09881=1208.273,266.119,-64.259,-176.887,6.849,148.355
C09882=1208.277,265.871,-64.232,-176.889,6.847,148.356
C09883=1208.281,265.622,-64.204,-176.891,6.845,148.356
C09884=1208.286,265.373,-64.177,-176.895,6.842,148.356
C09885=1208.290,265.125,-64.149,-176.897,6.840,148.356
C09886=1208.294,264.876,-64.122,-176.899,6.838,148.356
C09887=1208.299,264.628,-64.094,-176.902,6.835,148.356
C09888=1208.304,264.379,-64.067,-176.904,6.833,148.357
C09889=1208.309,264.131,-64.039,-176.907,6.831,148.357
C09890=1208.312,263.882,-64.011,-176.909,6.828,148.357
C09891=1208.317,263.634,-63.984,-176.912,6.826,148.357
C09892=1208.322,263.362,-63.955,-176.915,6.823,148.357
C09893=1208.327,263.089,-63.924,-176.917,6.821,148.358
C09894=1208.331,262.816,-63.894,-176.921,6.819,148.358
C09895=1208.336,262.543,-63.864,-176.923,6.816,148.358
C09896=1208.341,262.295,-63.837,-176.926,6.814,148.358
C09897=1208.345,262.046,-63.810,-176.928,6.812,148.358
C09898=1208.349,261.798,-63.782,-176.931,6.809,148.358
C09899=1208.354,261.549,-63.755,-176.933,6.807,148.359
C09900=1208.358,261.301,-63.727,-176.936,6.805,148.359
C09901=1208.363,261.052,-63.700,-176.938,6.803,148.359
C09902=1208.367,260.804,-63.673,-176.941,6.800,148.359
C09903=1208.371,260.555,-63.646,-176.943,6.798,148.359
C09904=1208.375,260.307,-63.619,-176.946,6.796,148.360
C09905=1208.380,260.058,-63.592,-176.949,6.793,148.360
C09906=1208.385,259.810,-63.565,-176.951,6.791,148.360
C09907=1208.389,259.562,-63.537,-176.954,6.789,148.360
C09908=1208.393,259.313,-63.509,-176.957,6.786,148.360
C09909=1208.398,259.064,-63.482,-176.959,6.784,148.360
C09910=1208.402,258.816,-63.455,-176.961,6.782,148.361
C09911=1208.407,258.567,-63.428,-176.964,6.780,148.361
C09912=1208.411,258.319,-63.402,-176.967,6.777,148.361
C09913=1208.416,258.071,-63.375,-176.969,6.775,148.361
C09914=1208.420,257.823,-63.347,-176.972,6.773,148.361
C09915=1208.424,257.574,-63.319,-176.974,6.770,148.361
C09916=1208.429,257.325,-63.292,-176.977,6.768,148.362
C09917=1208.433,257.077,-63.265,-176.979,6.766,148.362
C09918=1208.437,256.828,-63.239,-176.982,6.764,148.362
C09919=1208.442,256.580,-63.212,-176.984,6.761,148.362
C09920=1208.447,256.331,-63.185,-176.987,6.759,148.363
C09921=1208.451,256.083,-63.158,-176.989,6.757,148.363
C09922=1208.455,255.835,-63.131,-176.992,6.755,148.363
C09923=1208.459,255.586,-63.104,-176.994,6.752,148.363
C09924=1208.464,255.337,-63.077,-176.997,6.750,148.363
C09925=1208.469,255.089,-63.050,-176.999,6.748,148.363
C09926=1208.472,254.840,-63.023,-177.002,6.746,148.364
C09927=1208.477,254.592,-62.996,-177.005,6.744,148.364
C09928=1208.482,254.343,-62.969,-177.007,6.742,148.364
C09929=1208.487,254.094,-62.943,-177.010,6.740,148.364
C09930=1208.491,253.846,-62.916,-177.012,6.737,148.364
C09931=1208.495,253.598,-62.889,-177.015,6.735,148.365
C09932=1208.500,253.349,-62.862,-177.017,6.733,148.365
C09933=1208.504,253.101,-62.836,-177.020,6.731,148.365
C09934=1208.509,252.852,-62.809,-177.023,6.728,148.365
C09935=1208.513,252.604,-62.782,-177.025,6.726,148.365
C09936=1208.517,252.355,-62.754,-177.028,6.724,148.366
C09937=1208.522,252.106,-62.728,-177.030,6.722,148.366
C09938=1208.526,251.857,-62.701,-177.033,6.719,148.366
C09939=1208.530,251.609,-62.675,-177.035,6.717,148.366
C09940=1208.535,251.361,-62.648,-177.038,6.715,148.367
C09941=1208.539,251.112,-62.621,-177.040,6.713,148.367
C09942=1208.544,250.863,-62.595,-177.043,6.710,148.367
C09943=1208.548,250.615,-62.568,-177.045,6.708,148.367
C09944=1208.553,250.366,-62.541,-177.048,6.706,148.367
C09945=1208.557,250.118,-62.514,-177.051,6.704,148.368
C09946=1208.562,249.869,-62.488,-177.053,6.702,148.368
C09947=1208.566,249.621,-62.462,-177.056,6.700,148.368
C09948=1208.570,249.373,-62.435,-177.058,6.697,148.368
C09949=1208.575,249.123,-62.408,-177.061,6.695,148.368
C09950=1208.579,248.875,-62.382,-177.063,6.694,148.369
C09951=1208.584,248.627,-62.355,-177.066,6.691,148.369
C09952=1208.588,248.378,-62.329,-177.069,6.689,148.369
C09953=1208.593,248.129,-62.302,-177.071,6.687,148.369
C09954=1208.597,247.882,-62.276,-177.073,6.685,148.369
C09955=1208.602,247.633,-62.249,-177.076,6.683,148.370
C09956=1208.606,247.385,-62.223,-177.079,6.680,148.370
C09957=1208.611,247.136,-62.197,-177.081,6.678,148.370
C09958=1208.615,246.887,-62.170,-177.083,6.676,148.370
C09959=1208.620,246.639,-62.143,-177.086,6.674,148.371
C09960=1208.624,246.390,-62.117,-177.089,6.671,148.371
C09961=1208.629,246.142,-62.090,-177.091,6.669,148.371
C09962=1208.633,245.893,-62.065,-177.094,6.667,148.371
C09963=1208.638,245.644,-62.037,-177.096,6.665,148.371
C09964=1208.642,245.395,-62.012,-177.099,6.663,148.372
C09965=1208.646,245.147,-61.985,-177.102,6.661,148.372
C09966=1208.651,244.898,-61.959,-177.104,6.658,148.372
C09967=1208.655,244.650,-61.932,-177.107,6.656,148.372
C09968=1208.660,244.402,-61.906,-177.109,6.655,148.373
C09969=1208.664,244.153,-61.880,-177.112,6.652,148.373
C09970=1208.669,243.904,-61.854,-177.114,6.651,148.373
C09971=1208.673,243.656,-61.827,-177.117,6.648,148.373
C09972=1208.677,243.407,-61.801,-177.120,6.646,148.373
C09973=1208.682,243.158,-61.775,-177.122,6.644,148.374
C09974=1208.686,242.910,-61.749,-177.124,6.642,148.374
C09975=1208.691,242.661,-61.722,-177.127,6.640,148.374
C09976=1208.695,242.413,-61.696,-177.130,6.637,148.374
C09977=1208.700,242.165,-61.670,-177.132,6.635,148.374
C09978=1208.705,241.915,-61.644,-177.135,6.633,148.375
C09979=1208.709,241.667,-61.618,-177.137,6.631,148.375
C09980=1208.713,241.418,-61.592,-177.140,6.629,148.375
C09981=1208.718,241.169,-61.565,-177.142,6.627,148.376
C09982=1208.722,240.922,-61.539,-177.145,6.625,148.376
C09983=1208.727,240.673,-61.514,-177.148,6.622,148.376
C09984=1208.731,240.424,-61.487,-177.150,6.621,148.376
C09985=1208.736,240.175,-61.462,-177.153,6.619,148.377
C09986=1208.740,239.927,-61.435,-177.155,6.617,148.377
C09987=1208.745,239.678,-61.409,-177.158,6.615,148.377
C09988=1208.749,239.430,-61.383,-177.161,6.612,148.377
C09989=1208.754,239.181,-61.358,-177.163,6.610,148.377
C09990=1208.758,238.933,-61.331,-177.166,6.608,148.378
C09991=1208.763,238.684,-61.305,-177.168,6.606,148.378
C09992=1208.767,238.435,-61.279,-177.170,6.604,148.378
C09993=1208.772,238.187,-61.254,-177.173,6.602,148.378
C09994=1208.776,237.938,-61.228,-177.176,6.599,148.379
C09995=1208.780,237.689,-61.202,-177.178,6.597,148.379
C09996=1208.786,237.418,-61.173,-177.181,6.595,148.379
//INST
///DATE 2021/06/15 17:23
///ATTR SC,RW,RJ
////FRAME ROBOT
///GROUP1 RB1
NOP
MOVL C00000 V=800.0 PL=0
MOVL C00001 V=800.0 PL=0
MOVL C00002 V=800.0 PL=0
MOVL C00003 V=800.0 PL=0
MOVL C00004 V=800.0 PL=0
MOVL C00005 V=800.0 PL=0
MOVL C00006 V=800.0 PL=0
MOVL C00007 V=800.0 PL=0
MOVL C00008 V=800.0 PL=0
MOVL C00009 V=800.0 PL=0
MOVL C00010 V=800.0 PL=0
MOVL C00011 V=800.0 PL=0
MOVL C00012 V=800.0 PL=0
MOVL C00013 V=800.0 PL=0
MOVL C00014 V=800.0 PL=0
MOVL C00015 V=800.0 PL=0
MOVL C00016 V=800.0 PL=0
MOVL C00017 V=800.0 PL=0
MOVL C00018 V=800.0 PL=0
MOVL C00019 V=800.0 PL=0
MOVL C00020 V=800.0 PL=0
MOVL C00021 V=800.0 PL=0
MOVL C00022 V=800.0 PL=0
MOVL C00023 V=800.0 PL=0
MOVL C00024 V=800.0 PL=0
MOVL C00025 V=800.0 PL=0
MOVL C00026 V=800.0 PL=0
MOVL C00027 V=800.0 PL=0
MOVL C00028 V=800.0 PL=0
MOVL C00029 V=800.0 PL=0
MOVL C00030 V=800.0 PL=0
MOVL C00031 V=800.0 PL=0
MOVL C00032 V=800.0 PL=0
MOVL C00033 V=800.0 PL=0
MOVL C00034 V=800.0 PL=0
MOVL C00035 V=800.0 PL=0
MOVL C00036 V=800.0 PL=0
MOVL C00037 V=800.0 PL=0
MOVL C00038 V=800.0 PL=0
MOVL C00039 V=800.0 PL=0
MOVL C00040 V=800.0 PL=0
MOVL C00041 V=800.0 PL=0
MOVL C00042 V=800.0 PL=0
MOVL C00043 V=800.0 PL=0
MOVL C00044 V=800.0 PL=0
MOVL C00045 V=800.0 PL=0
MOVL C00046 V=800.0 PL=0
MOVL C00047 V=800.0 PL=0
MOVL C00048 V=800.0 PL=0
MOVL C00049 V=800.0 PL=0
MOVL C00050 V=800.0 PL=0
MOVL C00051 V=800.0 PL=0
MOVL C00052 V=800.0 PL=0
MOVL C00053 V=800.0 PL=0
MOVL C00054 V=800.0 PL=0
MOVL C00055 V=800.0 PL=0
MOVL C00056 V=800.0 PL=0
MOVL C00057 V=800.0 PL=0
MOVL C00058 V=800.0 PL=0
MOVL C00059 V=800.0 PL=0
MOVL C00060 V=800.0 PL=0
MOVL C00061 V=800.0 PL=0
MOVL C00062 V=800.0 PL=0
MOVL C00063 V=800.0 PL=0
MOVL C00064 V=800.0 PL=0
MOVL C00065 V=800.0 PL=0
MOVL C00066 V=800.0 PL=0
MOVL C00067 V=800.0 PL=0
MOVL C00068 V=800.0 PL=0
MOVL C00069 V=800.0 PL=0
MOVL C00070 V=800.0 PL=0
MOVL C00071 V=800.0 PL=0
MOVL C00072 V=800.0 PL=0
MOVL C00073 V=800.0 PL=0
MOVL C00074 V=800.0 PL=0
MOVL C00075 V=800.0 PL=0
MOVL C00076 V=800.0 PL=0
MOVL C00077 V=800.0 PL=0
MOVL C00078 V=800.0 PL=0
MOVL C00079 V=800.0 PL=0
MOVL C00080 V=800.0 PL=0
MOVL C00081 V=800.0 PL=0
MOVL C00082 V=800.0 PL=0
MOVL C00083 V=800.0 PL=0
MOVL C00084 V=800.0 PL=0
MOVL C00085 V=800.0 PL=0
MOVL C00086 V=800.0 PL=0
MOVL C00087 V=800.0 PL=0
MOVL C00088 V=800.0 PL=0
MOVL C00089 V=800.0 PL=0
MOVL C00090 V=800.0 PL=0
MOVL C00091 V=800.0 PL=0
MOVL C00092 V=800.0 PL=0
MOVL C00093 V=800.0 PL=0
MOVL C00094 V=800.0 PL=0
MOVL C00095 V=800.0 PL=0
MOVL C00096 V=800.0 PL=0
MOVL C00097 V=800.0 PL=0
MOVL C00098 V=800.0 PL=0
MOVL C00099 V=800.0 PL=0
MOVL C00100 V=800.0 PL=0
MOVL C00101 V=800.0 PL=0
MOVL C00102 V=800.0 PL=0
MOVL C00103 V=800.0 PL=0
MOVL C00104 V=800.0 PL=0
MOVL C00105 V=800.0 PL=0
MOVL C00106 V=800.0 PL=0
MOVL C00107 V=800.0 PL=0
MOVL C00108 V=800.0 PL=0
MOVL C00109 V=800.0 PL=0
MOVL C00110 V=800.0 PL=0
MOVL C00111 V=800.0 PL=0
MOVL C00112 V=800.0 PL=0
MOVL C00113 V=800.0 PL=0
MOVL C00114 V=800.0 PL=0
MOVL C00115 V=800.0 PL=0
MOVL C00116 V=800.0 PL=0
MOVL C00117 V=800.0 PL=0
MOVL C00118 V=800.0 PL=0
MOVL C00119 V=800.0 PL=0
MOVL C00120 V=800.0 PL=0
MOVL C00121 V=800.0 PL=0
MOVL C00122 V=800.0 PL=0
MOVL C00123 V=800.0 PL=0
MOVL C00124 V=800.0 PL=0
MOVL C00125 V=800.0 PL=0
MOVL C00126 V=800.0 PL=0
MOVL C00127 V=800.0 PL=0
MOVL C00128 V=800.0 PL=0
MOVL C00129 V=800.0 PL=0
MOVL C00130 V=800.0 PL=0
MOVL C00131 V=800.0 PL=0
MOVL C00132 V=800.0 PL=0
MOVL C00133 V=800.0 PL=0
MOVL C00134 V=800.0 PL=0
MOVL C00135 V=800.0 PL=0
MOVL C00136 V=800.0 PL=0
MOVL C00137 V=800.0 PL=0
MOVL C00138 V=800.0 PL=0
MOVL C00139 V=800.0 PL=0
MOVL C00140 V=800.0 PL=0
MOVL C00141 V=800.0 PL=0
MOVL C00142 V=800.0 PL=0
MOVL C00143 V=800.0 PL=0
MOVL C00144 V=800.0 PL=0
MOVL C00145 V=800.0 PL=0
MOVL C00146 V=800.0 PL=0
MOVL C00147 V=800.0 PL=0
MOVL C00148 V=800.0 PL=0
MOVL C00149 V=800.0 PL=0
MOVL C00150 V=800.0 PL=0
MOVL C00151 V=800.0 PL=0
MOVL C00152 V=800.0 PL=0
MOVL C00153 V=800.0 PL=0
MOVL C00154 V=800.0 PL=0
MOVL C00155 V=800.0 PL=0
MOVL C00156 V=800.0 PL=0
MOVL C00157 V=800.0 PL=0
MOVL C00158 V=800.0 PL=0
MOVL C00159 V=800.0 PL=0
MOVL C00160 V=800.0 PL=0
MOVL C00161 V=800.0 PL=0
MOVL C00162 V=800.0 PL=0
MOVL C00163 V=800.0 PL=0
MOVL C00164 V=800.0 PL=0
MOVL C00165 V=800.0 PL=0
MOVL C00166 V=800.0 PL=0
MOVL C00167 V=800.0 PL=0
MOVL C00168 V=800.0 PL=0
MOVL C00169 V=800.0 PL=0
MOVL C00170 V=800.0 PL=0
MOVL C00171 V=800.0 PL=0
MOVL C00172 V=800.0 PL=0
MOVL C00173 V=800.0 PL=0
MOVL C00174 V=800.0 PL=0
MOVL C00175 V=800.0 PL=0
MOVL C00176 V=800.0 PL=0
MOVL C00177 V=800.0 PL=0
MOVL C00178 V=800.0 PL=0
MOVL C00179 V=800.0 PL=0
MOVL C00180 V=800.0 PL=0
MOVL C00181 V=800.0 PL=0
MOVL C00182 V=800.0 PL=0
MOVL C00183 V=800.0 PL=0
MOVL C00184 V=800.0 PL=0
MOVL C00185 V=800.0 PL=0
MOVL C00186 V=800.0 PL=0
MOVL C00187 V=800.0 PL=0
MOVL C00188 V=800.0 PL=0
MOVL C00189 V=800.0 PL=0
MOVL C00190 V=800.0 PL=0
MOVL C00191 V=800.0 PL=0
MOVL C00192 V=800.0 PL=0
MOVL C00193 V=800.0 PL=0
MOVL C00194 V=800.0 PL=0
MOVL C00195 V=800.0 PL=0
MOVL C00196 V=800.0 PL=0
MOVL C00197 V=800.0 PL=0
MOVL C00198 V=800.0 PL=0
MOVL C00199 V=800.0 PL=0
MOVL C00200 V=800.0 PL=0
MOVL C00201 V=800.0 PL=0
MOVL C00202 V=800.0 PL=0
MOVL C00203 V=800.0 PL=0
MOVL C00204 V=800.0 PL=0
MOVL C00205 V=800.0 PL=0
MOVL C00206 V=800.0 PL=0
MOVL C00207 V=800.0 PL=0
MOVL C00208 V=800.0 PL=0
MOVL C00209 V=800.0 PL=0
MOVL C00210 V=800.0 PL=0
MOVL C00211 V=800.0 PL=0
MOVL C00212 V=800.0 PL=0
MOVL C00213 V=800.0 PL=0
MOVL C00214 V=800.0 PL=0
MOVL C00215 V=800.0 PL=0
MOVL C00216 V=800.0 PL=0
MOVL C00217 V=800.0 PL=0
MOVL C00218 V=800.0 PL=0
MOVL C00219 V=800.0 PL=0
MOVL C00220 V=800.0 PL=0
MOVL C00221 V=800.0 PL=0
MOVL C00222 V=800.0 PL=0
MOVL C00223 V=800.0 PL=0
MOVL C00224 V=800.0 PL=0
MOVL C00225 V=800.0 PL=0
MOVL C00226 V=800.0 PL=0
MOVL C00227 V=800.0 PL=0
MOVL C00228 V=800.0 PL=0
MOVL C00229 V=800.0 PL=0
MOVL C00230 V=800.0 PL=0
MOVL C00231 V=800.0 PL=0
MOVL C00232 V=800.0 PL=0
MOVL C00233 V=800.0 PL=0
MOVL C00234 V=800.0 PL=0
MOVL C00235 V=800.0 PL=0
MOVL C00236 V=800.0 PL=0
MOVL C00237 V=800.0 PL=0
MOVL C00238 V=800.0 PL=0
MOVL C00239 V=800.0 PL=0
MOVL C00240 V=800.0 PL=0
MOVL C00241 V=800.0 PL=0
MOVL C00242 V=800.0 PL=0
MOVL C00243 V=800.0 PL=0
MOVL C00244 V=800.0 PL=0
MOVL C00245 V=800.0 PL=0
MOVL C00246 V=800.0 PL=0
MOVL C00247 V=800.0 PL=0
MOVL C00248 V=800.0 PL=0
MOVL C00249 V=800.0 PL=0
MOVL C00250 V=800.0 PL=0
MOVL C00251 V=800.0 PL=0
MOVL C00252 V=800.0 PL=0
MOVL C00253 V=800.0 PL=0
MOVL C00254 V=800.0 PL=0
MOVL C00255 V=800.0 PL=0
MOVL C00256 V=800.0 PL=0
MOVL C00257 V=800.0 PL=0
MOVL C00258 V=800.0 PL=0
MOVL C00259 V=800.0 PL=0
MOVL C00260 V=800.0 PL=0
MOVL C00261 V=800.0 PL=0
MOVL C00262 V=800.0 PL=0
MOVL C00263 V=800.0 PL=0
MOVL C00264 V=800.0 PL=0
MOVL C00265 V=800.0 PL=0
MOVL C00266 V=800.0 PL=0
MOVL C00267 V=800.0 PL=0
MOVL C00268 V=800.0 PL=0
MOVL C00269 V=800.0 PL=0
MOVL C00270 V=800.0 PL=0
MOVL C00271 V=800.0 PL=0
MOVL C00272 V=800.0 PL=0
MOVL C00273 V=800.0 PL=0
MOVL C00274 V=800.0 PL=0
MOVL C00275 V=800.0 PL=0
MOVL C00276 V=800.0 PL=0
MOVL C00277 V=800.0 PL=0
MOVL C00278 V=800.0 PL=0
MOVL C00279 V=800.0 PL=0
MOVL C00280 V=800.0 PL=0
MOVL C00281 V=800.0 PL=0
MOVL C00282 V=800.0 PL=0
MOVL C00283 V=800.0 PL=0
MOVL C00284 V=800.0 PL=0
MOVL C00285 V=800.0 PL=0
MOVL C00286 V=800.0 PL=0
MOVL C00287 V=800.0 PL=0
MOVL C00288 V=800.0 PL=0
MOVL C00289 V=800.0 PL=0
MOVL C00290 V=800.0 PL=0
MOVL C00291 V=800.0 PL=0
MOVL C00292 V=800.0 PL=0
MOVL C00293 V=800.0 PL=0
MOVL C00294 V=800.0 PL=0
MOVL C00295 V=800.0 PL=0
MOVL C00296 V=800.0 PL=0
MOVL C00297 V=800.0 PL=0
MOVL C00298 V=800.0 PL=0
MOVL C00299 V=800.0 PL=0
MOVL C00300 V=800.0 PL=0
MOVL C00301 V=800.0 PL=0
MOVL C00302 V=800.0 PL=0
MOVL C00303 V=800.0 PL=0
MOVL C00304 V=800.0 PL=0
MOVL C00305 V=800.0 PL=0
MOVL C00306 V=800.0 PL=0
MOVL C00307 V=800.0 PL=0
MOVL C00308 V=800.0 PL=0
MOVL C00309 V=800.0 PL=0
MOVL C00310 V=800.0 PL=0
MOVL C00311 V=800.0 PL=0
MOVL C00312 V=800.0 PL=0
MOVL C00313 V=800.0 PL=0
MOVL C00314 V=800.0 PL=0
MOVL C00315 V=800.0 PL=0
MOVL C00316 V=800.0 PL=0
MOVL C00317 V=800.0 PL=0
MOVL C00318 V=800.0 PL=0
MOVL C00319 V=800.0 PL=0
MOVL C00320 V=800.0 PL=0
MOVL C00321 V=800.0 PL=0
MOVL C00322 V=800.0 PL=0
MOVL C00323 V=800.0 PL=0
MOVL C00324 V=800.0 PL=0
MOVL C00325 V=800.0 PL=0
MOVL C00326 V=800.0 PL=0
MOVL C00327 V=800.0 PL=0
MOVL C00328 V=800.0 PL=0
MOVL C00329 V=800.0 PL=0
MOVL C00330 V=800.0 PL=0
MOVL C00331 V=800.0 PL=0
MOVL C00332 V=800.0 PL=0
MOVL C00333 V=800.0 PL=0
MOVL C00334 V=800.0 PL=0
MOVL C00335 V=800.0 PL=0
MOVL C00336 V=800.0 PL=0
MOVL C00337 V=800.0 PL=0
MOVL C00338 V=800.0 PL=0
MOVL C00339 V=800.0 PL=0
MOVL C00340 V=800.0 PL=0
MOVL C00341 V=800.0 PL=0
MOVL C00342 V=800.0 PL=0
MOVL C00343 V=800.0 PL=0
MOVL C00344 V=800.0 PL=0
MOVL C00345 V=800.0 PL=0
MOVL C00346 V=800.0 PL=0
MOVL C00347 V=800.0 PL=0
MOVL C00348 V=800.0 PL=0
MOVL C00349 V=800.0 PL=0
MOVL C00350 V=800.0 PL=0
MOVL C00351 V=800.0 PL=0
MOVL C00352 V=800.0 PL=0
MOVL C00353 V=800.0 PL=0
MOVL C00354 V=800.0 PL=0
MOVL C00355 V=800.0 PL=0
MOVL C00356 V=800.0 PL=0
MOVL C00357 V=800.0 PL=0
MOVL C00358 V=800.0 PL=0
MOVL C00359 V=800.0 PL=0
MOVL C00360 V=800.0 PL=0
MOVL C00361 V=800.0 PL=0
MOVL C00362 V=800.0 PL=0
MOVL C00363 V=800.0 PL=0
MOVL C00364 V=800.0 PL=0
MOVL C00365 V=800.0 PL=0
MOVL C00366 V=800.0 PL=0
MOVL C00367 V=800.0 PL=0
MOVL C00368 V=800.0 PL=0
MOVL C00369 V=800.0 PL=0
MOVL C00370 V=800.0 PL=0
MOVL C00371 V=800.0 PL=0
MOVL C00372 V=800.0 PL=0
MOVL C00373 V=800.0 PL=0
MOVL C00374 V=800.0 PL=0
MOVL C00375 V=800.0 PL=0
MOVL C00376 V=800.0 PL=0
MOVL C00377 V=800.0 PL=0
MOVL C00378 V=800.0 PL=0
MOVL C00379 V=800.0 PL=0
MOVL C00380 V=800.0 PL=0
MOVL C00381 V=800.0 PL=0
MOVL C00382 V=800.0 PL=0
MOVL C00383 V=800.0 PL=0
MOVL C00384 V=800.0 PL=0
MOVL C00385 V=800.0 PL=0
MOVL C00386 V=800.0 PL=0
MOVL C00387 V=800.0 PL=0
MOVL C00388 V=800.0 PL=0
MOVL C00389 V=800.0 PL=0
MOVL C00390 V=800.0 PL=0
MOVL C00391 V=800.0 PL=0
MOVL C00392 V=800.0 PL=0
MOVL C00393 V=800.0 PL=0
MOVL C00394 V=800.0 PL=0
MOVL C00395 V=800.0 PL=0
MOVL C00396 V=800.0 PL=0
MOVL C00397 V=800.0 PL=0
MOVL C00398 V=800.0 PL=0
MOVL C00399 V=800.0 PL=0
MOVL C00400 V=800.0 PL=0
MOVL C00401 V=800.0 PL=0
MOVL C00402 V=800.0 PL=0
MOVL C00403 V=800.0 PL=0
MOVL C00404 V=800.0 PL=0
MOVL C00405 V=800.0 PL=0
MOVL C00406 V=800.0 PL=0
MOVL C00407 V=800.0 PL=0
MOVL C00408 V=800.0 PL=0
MOVL C00409 V=800.0 PL=0
MOVL C00410 V=800.0 PL=0
MOVL C00411 V=800.0 PL=0
MOVL C00412 V=800.0 PL=0
MOVL C00413 V=800.0 PL=0
MOVL C00414 V=800.0 PL=0
MOVL C00415 V=800.0 PL=0
MOVL C00416 V=800.0 PL=0
MOVL C00417 V=800.0 PL=0
MOVL C00418 V=800.0 PL=0
MOVL C00419 V=800.0 PL=0
MOVL C00420 V=800.0 PL=0
MOVL C00421 V=800.0 PL=0
MOVL C00422 V=800.0 PL=0
MOVL C00423 V=800.0 PL=0
MOVL C00424 V=800.0 PL=0
MOVL C00425 V=800.0 PL=0
MOVL C00426 V=800.0 PL=0
MOVL C00427 V=800.0 PL=0
MOVL C00428 V=800.0 PL=0
MOVL C00429 V=800.0 PL=0
MOVL C00430 V=800.0 PL=0
MOVL C00431 V=800.0 PL=0
MOVL C00432 V=800.0 PL=0
MOVL C00433 V=800.0 PL=0
MOVL C00434 V=800.0 PL=0
MOVL C00435 V=800.0 PL=0
MOVL C00436 V=800.0 PL=0
MOVL C00437 V=800.0 PL=0
MOVL C00438 V=800.0 PL=0
MOVL C00439 V=800.0 PL=0
MOVL C00440 V=800.0 PL=0
MOVL C00441 V=800.0 PL=0
MOVL C00442 V=800.0 PL=0
MOVL C00443 V=800.0 PL=0
MOVL C00444 V=800.0 PL=0
MOVL C00445 V=800.0 PL=0
MOVL C00446 V=800.0 PL=0
MOVL C00447 V=800.0 PL=0
MOVL C00448 V=800.0 PL=0
MOVL C00449 V=800.0 PL=0
MOVL C00450 V=800.0 PL=0
MOVL C00451 V=800.0 PL=0
MOVL C00452 V=800.0 PL=0
MOVL C00453 V=800.0 PL=0
MOVL C00454 V=800.0 PL=0
MOVL C00455 V=800.0 PL=0
MOVL C00456 V=800.0 PL=0
MOVL C00457 V=800.0 PL=0
MOVL C00458 V=800.0 PL=0
MOVL C00459 V=800.0 PL=0
MOVL C00460 V=800.0 PL=0
MOVL C00461 V=800.0 PL=0
MOVL C00462 V=800.0 PL=0
MOVL C00463 V=800.0 PL=0
MOVL C00464 V=800.0 PL=0
MOVL C00465 V=800.0 PL=0
MOVL C00466 V=800.0 PL=0
MOVL C00467 V=800.0 PL=0
MOVL C00468 V=800.0 PL=0
MOVL C00469 V=800.0 PL=0
MOVL C00470 V=800.0 PL=0
MOVL C00471 V=800.0 PL=0
MOVL C00472 V=800.0 PL=0
MOVL C00473 V=800.0 PL=0
MOVL C00474 V=800.0 PL=0
MOVL C00475 V=800.0 PL=0
MOVL C00476 V=800.0 PL=0
MOVL C00477 V=800.0 PL=0
MOVL C00478 V=800.0 PL=0
MOVL C00479 V=800.0 PL=0
MOVL C00480 V=800.0 PL=0
MOVL C00481 V=800.0 PL=0
MOVL C00482 V=800.0 PL=0
MOVL C00483 V=800.0 PL=0
MOVL C00484 V=800.0 PL=0
MOVL C00485 V=800.0 PL=0
MOVL C00486 V=800.0 PL=0
MOVL C00487 V=800.0 PL=0
MOVL C00488 V=800.0 PL=0
MOVL C00489 V=800.0 PL=0
MOVL C00490 V=800.0 PL=0
MOVL C00491 V=800.0 PL=0
MOVL C00492 V=800.0 PL=0
MOVL C00493 V=800.0 PL=0
MOVL C00494 V=800.0 PL=0
MOVL C00495 V=800.0 PL=0
MOVL C00496 V=800.0 PL=0
MOVL C00497 V=800.0 PL=0
MOVL C00498 V=800.0 PL=0
MOVL C00499 V=800.0 PL=0
MOVL C00500 V=800.0 PL=0
MOVL C00501 V=800.0 PL=0
MOVL C00502 V=800.0 PL=0
MOVL C00503 V=800.0 PL=0
MOVL C00504 V=800.0 PL=0
MOVL C00505 V=800.0 PL=0
MOVL C00506 V=800.0 PL=0
MOVL C00507 V=800.0 PL=0
MOVL C00508 V=800.0 PL=0
MOVL C00509 V=800.0 PL=0
MOVL C00510 V=800.0 PL=0
MOVL C00511 V=800.0 PL=0
MOVL C00512 V=800.0 PL=0
MOVL C00513 V=800.0 PL=0
MOVL C00514 V=800.0 PL=0
MOVL C00515 V=800.0 PL=0
MOVL C00516 V=800.0 PL=0
MOVL C00517 V=800.0 PL=0
MOVL C00518 V=800.0 PL=0
MOVL C00519 V=800.0 PL=0
MOVL C00520 V=800.0 PL=0
MOVL C00521 V=800.0 PL=0
MOVL C00522 V=800.0 PL=0
MOVL C00523 V=800.0 PL=0
MOVL C00524 V=800.0 PL=0
MOVL C00525 V=800.0 PL=0
MOVL C00526 V=800.0 PL=0
MOVL C00527 V=800.0 PL=0
MOVL C00528 V=800.0 PL=0
MOVL C00529 V=800.0 PL=0
MOVL C00530 V=800.0 PL=0
MOVL C00531 V=800.0 PL=0
MOVL C00532 V=800.0 PL=0
MOVL C00533 V=800.0 PL=0
MOVL C00534 V=800.0 PL=0
MOVL C00535 V=800.0 PL=0
MOVL C00536 V=800.0 PL=0
MOVL C00537 V=800.0 PL=0
MOVL C00538 V=800.0 PL=0
MOVL C00539 V=800.0 PL=0
MOVL C00540 V=800.0 PL=0
MOVL C00541 V=800.0 PL=0
MOVL C00542 V=800.0 PL=0
MOVL C00543 V=800.0 PL=0
MOVL C00544 V=800.0 PL=0
MOVL C00545 V=800.0 PL=0
MOVL C00546 V=800.0 PL=0
MOVL C00547 V=800.0 PL=0
MOVL C00548 V=800.0 PL=0
MOVL C00549 V=800.0 PL=0
MOVL C00550 V=800.0 PL=0
MOVL C00551 V=800.0 PL=0
MOVL C00552 V=800.0 PL=0
MOVL C00553 V=800.0 PL=0
MOVL C00554 V=800.0 PL=0
MOVL C00555 V=800.0 PL=0
MOVL C00556 V=800.0 PL=0
MOVL C00557 V=800.0 PL=0
MOVL C00558 V=800.0 PL=0
MOVL C00559 V=800.0 PL=0
MOVL C00560 V=800.0 PL=0
MOVL C00561 V=800.0 PL=0
MOVL C00562 V=800.0 PL=0
MOVL C00563 V=800.0 PL=0
MOVL C00564 V=800.0 PL=0
MOVL C00565 V=800.0 PL=0
MOVL C00566 V=800.0 PL=0
MOVL C00567 V=800.0 PL=0
MOVL C00568 V=800.0 PL=0
MOVL C00569 V=800.0 PL=0
MOVL C00570 V=800.0 PL=0
MOVL C00571 V=800.0 PL=0
MOVL C00572 V=800.0 PL=0
MOVL C00573 V=800.0 PL=0
MOVL C00574 V=800.0 PL=0
MOVL C00575 V=800.0 PL=0
MOVL C00576 V=800.0 PL=0
MOVL C00577 V=800.0 PL=0
MOVL C00578 V=800.0 PL=0
MOVL C00579 V=800.0 PL=0
MOVL C00580 V=800.0 PL=0
MOVL C00581 V=800.0 PL=0
MOVL C00582 V=800.0 PL=0
MOVL C00583 V=800.0 PL=0
MOVL C00584 V=800.0 PL=0
MOVL C00585 V=800.0 PL=0
MOVL C00586 V=800.0 PL=0
MOVL C00587 V=800.0 PL=0
MOVL C00588 V=800.0 PL=0
MOVL C00589 V=800.0 PL=0
MOVL C00590 V=800.0 PL=0
MOVL C00591 V=800.0 PL=0
MOVL C00592 V=800.0 PL=0
MOVL C00593 V=800.0 PL=0
MOVL C00594 V=800.0 PL=0
MOVL C00595 V=800.0 PL=0
MOVL C00596 V=800.0 PL=0
MOVL C00597 V=800.0 PL=0
MOVL C00598 V=800.0 PL=0
MOVL C00599 V=800.0 PL=0
MOVL C00600 V=800.0 PL=0
MOVL C00601 V=800.0 PL=0
MOVL C00602 V=800.0 PL=0
MOVL C00603 V=800.0 PL=0
MOVL C00604 V=800.0 PL=0
MOVL C00605 V=800.0 PL=0
MOVL C00606 V=800.0 PL=0
MOVL C00607 V=800.0 PL=0
MOVL C00608 V=800.0 PL=0
MOVL C00609 V=800.0 PL=0
MOVL C00610 V=800.0 PL=0
MOVL C00611 V=800.0 PL=0
MOVL C00612 V=800.0 PL=0
MOVL C00613 V=800.0 PL=0
MOVL C00614 V=800.0 PL=0
MOVL C00615 V=800.0 PL=0
MOVL C00616 V=800.0 PL=0
MOVL C00617 V=800.0 PL=0
MOVL C00618 V=800.0 PL=0
MOVL C00619 V=800.0 PL=0
MOVL C00620 V=800.0 PL=0
MOVL C00621 V=800.0 PL=0
MOVL C00622 V=800.0 PL=0
MOVL C00623 V=800.0 PL=0
MOVL C00624 V=800.0 PL=0
MOVL C00625 V=800.0 PL=0
MOVL C00626 V=800.0 PL=0
MOVL C00627 V=800.0 PL=0
MOVL C00628 V=800.0 PL=0
MOVL C00629 V=800.0 PL=0
MOVL C00630 V=800.0 PL=0
MOVL C00631 V=800.0 PL=0
MOVL C00632 V=800.0 PL=0
MOVL C00633 V=800.0 PL=0
MOVL C00634 V=800.0 PL=0
MOVL C00635 V=800.0 PL=0
MOVL C00636 V=800.0 PL=0
MOVL C00637 V=800.0 PL=0
MOVL C00638 V=800.0 PL=0
MOVL C00639 V=800.0 PL=0
MOVL C00640 V=800.0 PL=0
MOVL C00641 V=800.0 PL=0
MOVL C00642 V=800.0 PL=0
MOVL C00643 V=800.0 PL=0
MOVL C00644 V=800.0 PL=0
MOVL C00645 V=800.0 PL=0
MOVL C00646 V=800.0 PL=0
MOVL C00647 V=800.0 PL=0
MOVL C00648 V=800.0 PL=0
MOVL C00649 V=800.0 PL=0
MOVL C00650 V=800.0 PL=0
MOVL C00651 V=800.0 PL=0
MOVL C00652 V=800.0 PL=0
MOVL C00653 V=800.0 PL=0
MOVL C00654 V=800.0 PL=0
MOVL C00655 V=800.0 PL=0
MOVL C00656 V=800.0 PL=0
MOVL C00657 V=800.0 PL=0
MOVL C00658 V=800.0 PL=0
MOVL C00659 V=800.0 PL=0
MOVL C00660 V=800.0 PL=0
MOVL C00661 V=800.0 PL=0
MOVL C00662 V=800.0 PL=0
MOVL C00663 V=800.0 PL=0
MOVL C00664 V=800.0 PL=0
MOVL C00665 V=800.0 PL=0
MOVL C00666 V=800.0 PL=0
MOVL C00667 V=800.0 PL=0
MOVL C00668 V=800.0 PL=0
MOVL C00669 V=800.0 PL=0
MOVL C00670 V=800.0 PL=0
MOVL C00671 V=800.0 PL=0
MOVL C00672 V=800.0 PL=0
MOVL C00673 V=800.0 PL=0
MOVL C00674 V=800.0 PL=0
MOVL C00675 V=800.0 PL=0
MOVL C00676 V=800.0 PL=0
MOVL C00677 V=800.0 PL=0
MOVL C00678 V=800.0 PL=0
MOVL C00679 V=800.0 PL=0
MOVL C00680 V=800.0 PL=0
MOVL C00681 V=800.0 PL=0
MOVL C00682 V=800.0 PL=0
MOVL C00683 V=800.0 PL=0
MOVL C00684 V=800.0 PL=0
MOVL C00685 V=800.0 PL=0
MOVL C00686 V=800.0 PL=0
MOVL C00687 V=800.0 PL=0
MOVL C00688 V=800.0 PL=0
MOVL C00689 V=800.0 PL=0
MOVL C00690 V=800.0 PL=0
MOVL C00691 V=800.0 PL=0
MOVL C00692 V=800.0 PL=0
MOVL C00693 V=800.0 PL=0
MOVL C00694 V=800.0 PL=0
MOVL C00695 V=800.0 PL=0
MOVL C00696 V=800.0 PL=0
MOVL C00697 V=800.0 PL=0
MOVL C00698 V=800.0 PL=0
MOVL C00699 V=800.0 PL=0
MOVL C00700 V=800.0 PL=0
MOVL C00701 V=800.0 PL=0
MOVL C00702 V=800.0 PL=0
MOVL C00703 V=800.0 PL=0
MOVL C00704 V=800.0 PL=0
MOVL C00705 V=800.0 PL=0
MOVL C00706 V=800.0 PL=0
MOVL C00707 V=800.0 PL=0
MOVL C00708 V=800.0 PL=0
MOVL C00709 V=800.0 PL=0
MOVL C00710 V=800.0 PL=0
MOVL C00711 V=800.0 PL=0
MOVL C00712 V=800.0 PL=0
MOVL C00713 V=800.0 PL=0
MOVL C00714 V=800.0 PL=0
MOVL C00715 V=800.0 PL=0
MOVL C00716 V=800.0 PL=0
MOVL C00717 V=800.0 PL=0
MOVL C00718 V=800.0 PL=0
MOVL C00719 V=800.0 PL=0
MOVL C00720 V=800.0 PL=0
MOVL C00721 V=800.0 PL=0
MOVL C00722 V=800.0 PL=0
MOVL C00723 V=800.0 PL=0
MOVL C00724 V=800.0 PL=0
MOVL C00725 V=800.0 PL=0
MOVL C00726 V=800.0 PL=0
MOVL C00727 V=800.0 PL=0
MOVL C00728 V=800.0 PL=0
MOVL C00729 V=800.0 PL=0
MOVL C00730 V=800.0 PL=0
MOVL C00731 V=800.0 PL=0
MOVL C00732 V=800.0 PL=0
MOVL C00733 V=800.0 PL=0
MOVL C00734 V=800.0 PL=0
MOVL C00735 V=800.0 PL=0
MOVL C00736 V=800.0 PL=0
MOVL C00737 V=800.0 PL=0
MOVL C00738 V=800.0 PL=0
MOVL C00739 V=800.0 PL=0
MOVL C00740 V=800.0 PL=0
MOVL C00741 V=800.0 PL=0
MOVL C00742 V=800.0 PL=0
MOVL C00743 V=800.0 PL=0
MOVL C00744 V=800.0 PL=0
MOVL C00745 V=800.0 PL=0
MOVL C00746 V=800.0 PL=0
MOVL C00747 V=800.0 PL=0
MOVL C00748 V=800.0 PL=0
MOVL C00749 V=800.0 PL=0
MOVL C00750 V=800.0 PL=0
MOVL C00751 V=800.0 PL=0
MOVL C00752 V=800.0 PL=0
MOVL C00753 V=800.0 PL=0
MOVL C00754 V=800.0 PL=0
MOVL C00755 V=800.0 PL=0
MOVL C00756 V=800.0 PL=0
MOVL C00757 V=800.0 PL=0
MOVL C00758 V=800.0 PL=0
MOVL C00759 V=800.0 PL=0
MOVL C00760 V=800.0 PL=0
MOVL C00761 V=800.0 PL=0
MOVL C00762 V=800.0 PL=0
MOVL C00763 V=800.0 PL=0
MOVL C00764 V=800.0 PL=0
MOVL C00765 V=800.0 PL=0
MOVL C00766 V=800.0 PL=0
MOVL C00767 V=800.0 PL=0
MOVL C00768 V=800.0 PL=0
MOVL C00769 V=800.0 PL=0
MOVL C00770 V=800.0 PL=0
MOVL C00771 V=800.0 PL=0
MOVL C00772 V=800.0 PL=0
MOVL C00773 V=800.0 PL=0
MOVL C00774 V=800.0 PL=0
MOVL C00775 V=800.0 PL=0
MOVL C00776 V=800.0 PL=0
MOVL C00777 V=800.0 PL=0
MOVL C00778 V=800.0 PL=0
MOVL C00779 V=800.0 PL=0
MOVL C00780 V=800.0 PL=0
MOVL C00781 V=800.0 PL=0
MOVL C00782 V=800.0 PL=0
MOVL C00783 V=800.0 PL=0
MOVL C00784 V=800.0 PL=0
MOVL C00785 V=800.0 PL=0
MOVL C00786 V=800.0 PL=0
MOVL C00787 V=800.0 PL=0
MOVL C00788 V=800.0 PL=0
MOVL C00789 V=800.0 PL=0
MOVL C00790 V=800.0 PL=0
MOVL C00791 V=800.0 PL=0
MOVL C00792 V=800.0 PL=0
MOVL C00793 V=800.0 PL=0
MOVL C00794 V=800.0 PL=0
MOVL C00795 V=800.0 PL=0
MOVL C00796 V=800.0 PL=0
MOVL C00797 V=800.0 PL=0
MOVL C00798 V=800.0 PL=0
MOVL C00799 V=800.0 PL=0
MOVL C00800 V=800.0 PL=0
MOVL C00801 V=800.0 PL=0
MOVL C00802 V=800.0 PL=0
MOVL C00803 V=800.0 PL=0
MOVL C00804 V=800.0 PL=0
MOVL C00805 V=800.0 PL=0
MOVL C00806 V=800.0 PL=0
MOVL C00807 V=800.0 PL=0
MOVL C00808 V=800.0 PL=0
MOVL C00809 V=800.0 PL=0
MOVL C00810 V=800.0 PL=0
MOVL C00811 V=800.0 PL=0
MOVL C00812 V=800.0 PL=0
MOVL C00813 V=800.0 PL=0
MOVL C00814 V=800.0 PL=0
MOVL C00815 V=800.0 PL=0
MOVL C00816 V=800.0 PL=0
MOVL C00817 V=800.0 PL=0
MOVL C00818 V=800.0 PL=0
MOVL C00819 V=800.0 PL=0
MOVL C00820 V=800.0 PL=0
MOVL C00821 V=800.0 PL=0
MOVL C00822 V=800.0 PL=0
MOVL C00823 V=800.0 PL=0
MOVL C00824 V=800.0 PL=0
MOVL C00825 V=800.0 PL=0
MOVL C00826 V=800.0 PL=0
MOVL C00827 V=800.0 PL=0
MOVL C00828 V=800.0 PL=0
MOVL C00829 V=800.0 PL=0
MOVL C00830 V=800.0 PL=0
MOVL C00831 V=800.0 PL=0
MOVL C00832 V=800.0 PL=0
MOVL C00833 V=800.0 PL=0
MOVL C00834 V=800.0 PL=0
MOVL C00835 V=800.0 PL=0
MOVL C00836 V=800.0 PL=0
MOVL C00837 V=800.0 PL=0
MOVL C00838 V=800.0 PL=0
MOVL C00839 V=800.0 PL=0
MOVL C00840 V=800.0 PL=0
MOVL C00841 V=800.0 PL=0
MOVL C00842 V=800.0 PL=0
MOVL C00843 V=800.0 PL=0
MOVL C00844 V=800.0 PL=0
MOVL C00845 V=800.0 PL=0
MOVL C00846 V=800.0 PL=0
MOVL C00847 V=800.0 PL=0
MOVL C00848 V=800.0 PL=0
MOVL C00849 V=800.0 PL=0
MOVL C00850 V=800.0 PL=0
MOVL C00851 V=800.0 PL=0
MOVL C00852 V=800.0 PL=0
MOVL C00853 V=800.0 PL=0
MOVL C00854 V=800.0 PL=0
MOVL C00855 V=800.0 PL=0
MOVL C00856 V=800.0 PL=0
MOVL C00857 V=800.0 PL=0
MOVL C00858 V=800.0 PL=0
MOVL C00859 V=800.0 PL=0
MOVL C00860 V=800.0 PL=0
MOVL C00861 V=800.0 PL=0
MOVL C00862 V=800.0 PL=0
MOVL C00863 V=800.0 PL=0
MOVL C00864 V=800.0 PL=0
MOVL C00865 V=800.0 PL=0
MOVL C00866 V=800.0 PL=0
MOVL C00867 V=800.0 PL=0
MOVL C00868 V=800.0 PL=0
MOVL C00869 V=800.0 PL=0
MOVL C00870 V=800.0 PL=0
MOVL C00871 V=800.0 PL=0
MOVL C00872 V=800.0 PL=0
MOVL C00873 V=800.0 PL=0
MOVL C00874 V=800.0 PL=0
MOVL C00875 V=800.0 PL=0
MOVL C00876 V=800.0 PL=0
MOVL C00877 V=800.0 PL=0
MOVL C00878 V=800.0 PL=0
MOVL C00879 V=800.0 PL=0
MOVL C00880 V=800.0 PL=0
MOVL C00881 V=800.0 PL=0
MOVL C00882 V=800.0 PL=0
MOVL C00883 V=800.0 PL=0
MOVL C00884 V=800.0 PL=0
MOVL C00885 V=800.0 PL=0
MOVL C00886 V=800.0 PL=0
MOVL C00887 V=800.0 PL=0
MOVL C00888 V=800.0 PL=0
MOVL C00889 V=800.0 PL=0
MOVL C00890 V=800.0 PL=0
MOVL C00891 V=800.0 PL=0
MOVL C00892 V=800.0 PL=0
MOVL C00893 V=800.0 PL=0
MOVL C00894 V=800.0 PL=0
MOVL C00895 V=800.0 PL=0
MOVL C00896 V=800.0 PL=0
MOVL C00897 V=800.0 PL=0
MOVL C00898 V=800.0 PL=0
MOVL C00899 V=800.0 PL=0
MOVL C00900 V=800.0 PL=0
MOVL C00901 V=800.0 PL=0
MOVL C00902 V=800.0 PL=0
MOVL C00903 V=800.0 PL=0
MOVL C00904 V=800.0 PL=0
MOVL C00905 V=800.0 PL=0
MOVL C00906 V=800.0 PL=0
MOVL C00907 V=800.0 PL=0
MOVL C00908 V=800.0 PL=0
MOVL C00909 V=800.0 PL=0
MOVL C00910 V=800.0 PL=0
MOVL C00911 V=800.0 PL=0
MOVL C00912 V=800.0 PL=0
MOVL C00913 V=800.0 PL=0
MOVL C00914 V=800.0 PL=0
MOVL C00915 V=800.0 PL=0
MOVL C00916 V=800.0 PL=0
MOVL C00917 V=800.0 PL=0
MOVL C00918 V=800.0 PL=0
MOVL C00919 V=800.0 PL=0
MOVL C00920 V=800.0 PL=0
MOVL C00921 V=800.0 PL=0
MOVL C00922 V=800.0 PL=0
MOVL C00923 V=800.0 PL=0
MOVL C00924 V=800.0 PL=0
MOVL C00925 V=800.0 PL=0
MOVL C00926 V=800.0 PL=0
MOVL C00927 V=800.0 PL=0
MOVL C00928 V=800.0 PL=0
MOVL C00929 V=800.0 PL=0
MOVL C00930 V=800.0 PL=0
MOVL C00931 V=800.0 PL=0
MOVL C00932 V=800.0 PL=0
MOVL C00933 V=800.0 PL=0
MOVL C00934 V=800.0 PL=0
MOVL C00935 V=800.0 PL=0
MOVL C00936 V=800.0 PL=0
MOVL C00937 V=800.0 PL=0
MOVL C00938 V=800.0 PL=0
MOVL C00939 V=800.0 PL=0
MOVL C00940 V=800.0 PL=0
MOVL C00941 V=800.0 PL=0
MOVL C00942 V=800.0 PL=0
MOVL C00943 V=800.0 PL=0
MOVL C00944 V=800.0 PL=0
MOVL C00945 V=800.0 PL=0
MOVL C00946 V=800.0 PL=0
MOVL C00947 V=800.0 PL=0
MOVL C00948 V=800.0 PL=0
MOVL C00949 V=800.0 PL=0
MOVL C00950 V=800.0 PL=0
MOVL C00951 V=800.0 PL=0
MOVL C00952 V=800.0 PL=0
MOVL C00953 V=800.0 PL=0
MOVL C00954 V=800.0 PL=0
MOVL C00955 V=800.0 PL=0
MOVL C00956 V=800.0 PL=0
MOVL C00957 V=800.0 PL=0
MOVL C00958 V=800.0 PL=0
MOVL C00959 V=800.0 PL=0
MOVL C00960 V=800.0 PL=0
MOVL C00961 V=800.0 PL=0
MOVL C00962 V=800.0 PL=0
MOVL C00963 V=800.0 PL=0
MOVL C00964 V=800.0 PL=0
MOVL C00965 V=800.0 PL=0
MOVL C00966 V=800.0 PL=0
MOVL C00967 V=800.0 PL=0
MOVL C00968 V=800.0 PL=0
MOVL C00969 V=800.0 PL=0
MOVL C00970 V=800.0 PL=0
MOVL C00971 V=800.0 PL=0
MOVL C00972 V=800.0 PL=0
MOVL C00973 V=800.0 PL=0
MOVL C00974 V=800.0 PL=0
MOVL C00975 V=800.0 PL=0
MOVL C00976 V=800.0 PL=0
MOVL C00977 V=800.0 PL=0
MOVL C00978 V=800.0 PL=0
MOVL C00979 V=800.0 PL=0
MOVL C00980 V=800.0 PL=0
MOVL C00981 V=800.0 PL=0
MOVL C00982 V=800.0 PL=0
MOVL C00983 V=800.0 PL=0
MOVL C00984 V=800.0 PL=0
MOVL C00985 V=800.0 PL=0
MOVL C00986 V=800.0 PL=0
MOVL C00987 V=800.0 PL=0
MOVL C00988 V=800.0 PL=0
MOVL C00989 V=800.0 PL=0
MOVL C00990 V=800.0 PL=0
MOVL C00991 V=800.0 PL=0
MOVL C00992 V=800.0 PL=0
MOVL C00993 V=800.0 PL=0
MOVL C00994 V=800.0 PL=0
MOVL C00995 V=800.0 PL=0
MOVL C00996 V=800.0 PL=0
MOVL C00997 V=800.0 PL=0
MOVL C00998 V=800.0 PL=0
MOVL C00999 V=800.0 PL=0
MOVL C01000 V=800.0 PL=0
MOVL C01001 V=800.0 PL=0
MOVL C01002 V=800.0 PL=0
MOVL C01003 V=800.0 PL=0
MOVL C01004 V=800.0 PL=0
MOVL C01005 V=800.0 PL=0
MOVL C01006 V=800.0 PL=0
MOVL C01007 V=800.0 PL=0
MOVL C01008 V=800.0 PL=0
MOVL C01009 V=800.0 PL=0
MOVL C01010 V=800.0 PL=0
MOVL C01011 V=800.0 PL=0
MOVL C01012 V=800.0 PL=0
MOVL C01013 V=800.0 PL=0
MOVL C01014 V=800.0 PL=0
MOVL C01015 V=800.0 PL=0
MOVL C01016 V=800.0 PL=0
MOVL C01017 V=800.0 PL=0
MOVL C01018 V=800.0 PL=0
MOVL C01019 V=800.0 PL=0
MOVL C01020 V=800.0 PL=0
MOVL C01021 V=800.0 PL=0
MOVL C01022 V=800.0 PL=0
MOVL C01023 V=800.0 PL=0
MOVL C01024 V=800.0 PL=0
MOVL C01025 V=800.0 PL=0
MOVL C01026 V=800.0 PL=0
MOVL C01027 V=800.0 PL=0
MOVL C01028 V=800.0 PL=0
MOVL C01029 V=800.0 PL=0
MOVL C01030 V=800.0 PL=0
MOVL C01031 V=800.0 PL=0
MOVL C01032 V=800.0 PL=0
MOVL C01033 V=800.0 PL=0
MOVL C01034 V=800.0 PL=0
MOVL C01035 V=800.0 PL=0
MOVL C01036 V=800.0 PL=0
MOVL C01037 V=800.0 PL=0
MOVL C01038 V=800.0 PL=0
MOVL C01039 V=800.0 PL=0
MOVL C01040 V=800.0 PL=0
MOVL C01041 V=800.0 PL=0
MOVL C01042 V=800.0 PL=0
MOVL C01043 V=800.0 PL=0
MOVL C01044 V=800.0 PL=0
MOVL C01045 V=800.0 PL=0
MOVL C01046 V=800.0 PL=0
MOVL C01047 V=800.0 PL=0
MOVL C01048 V=800.0 PL=0
MOVL C01049 V=800.0 PL=0
MOVL C01050 V=800.0 PL=0
MOVL C01051 V=800.0 PL=0
MOVL C01052 V=800.0 PL=0
MOVL C01053 V=800.0 PL=0
MOVL C01054 V=800.0 PL=0
MOVL C01055 V=800.0 PL=0
MOVL C01056 V=800.0 PL=0
MOVL C01057 V=800.0 PL=0
MOVL C01058 V=800.0 PL=0
MOVL C01059 V=800.0 PL=0
MOVL C01060 V=800.0 PL=0
MOVL C01061 V=800.0 PL=0
MOVL C01062 V=800.0 PL=0
MOVL C01063 V=800.0 PL=0
MOVL C01064 V=800.0 PL=0
MOVL C01065 V=800.0 PL=0
MOVL C01066 V=800.0 PL=0
MOVL C01067 V=800.0 PL=0
MOVL C01068 V=800.0 PL=0
MOVL C01069 V=800.0 PL=0
MOVL C01070 V=800.0 PL=0
MOVL C01071 V=800.0 PL=0
MOVL C01072 V=800.0 PL=0
MOVL C01073 V=800.0 PL=0
MOVL C01074 V=800.0 PL=0
MOVL C01075 V=800.0 PL=0
MOVL C01076 V=800.0 PL=0
MOVL C01077 V=800.0 PL=0
MOVL C01078 V=800.0 PL=0
MOVL C01079 V=800.0 PL=0
MOVL C01080 V=800.0 PL=0
MOVL C01081 V=800.0 PL=0
MOVL C01082 V=800.0 PL=0
MOVL C01083 V=800.0 PL=0
MOVL C01084 V=800.0 PL=0
MOVL C01085 V=800.0 PL=0
MOVL C01086 V=800.0 PL=0
MOVL C01087 V=800.0 PL=0
MOVL C01088 V=800.0 PL=0
MOVL C01089 V=800.0 PL=0
MOVL C01090 V=800.0 PL=0
MOVL C01091 V=800.0 PL=0
MOVL C01092 V=800.0 PL=0
MOVL C01093 V=800.0 PL=0
MOVL C01094 V=800.0 PL=0
MOVL C01095 V=800.0 PL=0
MOVL C01096 V=800.0 PL=0
MOVL C01097 V=800.0 PL=0
MOVL C01098 V=800.0 PL=0
MOVL C01099 V=800.0 PL=0
MOVL C01100 V=800.0 PL=0
MOVL C01101 V=800.0 PL=0
MOVL C01102 V=800.0 PL=0
MOVL C01103 V=800.0 PL=0
MOVL C01104 V=800.0 PL=0
MOVL C01105 V=800.0 PL=0
MOVL C01106 V=800.0 PL=0
MOVL C01107 V=800.0 PL=0
MOVL C01108 V=800.0 PL=0
MOVL C01109 V=800.0 PL=0
MOVL C01110 V=800.0 PL=0
MOVL C01111 V=800.0 PL=0
MOVL C01112 V=800.0 PL=0
MOVL C01113 V=800.0 PL=0
MOVL C01114 V=800.0 PL=0
MOVL C01115 V=800.0 PL=0
MOVL C01116 V=800.0 PL=0
MOVL C01117 V=800.0 PL=0
MOVL C01118 V=800.0 PL=0
MOVL C01119 V=800.0 PL=0
MOVL C01120 V=800.0 PL=0
MOVL C01121 V=800.0 PL=0
MOVL C01122 V=800.0 PL=0
MOVL C01123 V=800.0 PL=0
MOVL C01124 V=800.0 PL=0
MOVL C01125 V=800.0 PL=0
MOVL C01126 V=800.0 PL=0
MOVL C01127 V=800.0 PL=0
MOVL C01128 V=800.0 PL=0
MOVL C01129 V=800.0 PL=0
MOVL C01130 V=800.0 PL=0
MOVL C01131 V=800.0 PL=0
MOVL C01132 V=800.0 PL=0
MOVL C01133 V=800.0 PL=0
MOVL C01134 V=800.0 PL=0
MOVL C01135 V=800.0 PL=0
MOVL C01136 V=800.0 PL=0
MOVL C01137 V=800.0 PL=0
MOVL C01138 V=800.0 PL=0
MOVL C01139 V=800.0 PL=0
MOVL C01140 V=800.0 PL=0
MOVL C01141 V=800.0 PL=0
MOVL C01142 V=800.0 PL=0
MOVL C01143 V=800.0 PL=0
MOVL C01144 V=800.0 PL=0
MOVL C01145 V=800.0 PL=0
MOVL C01146 V=800.0 PL=0
MOVL C01147 V=800.0 PL=0
MOVL C01148 V=800.0 PL=0
MOVL C01149 V=800.0 PL=0
MOVL C01150 V=800.0 PL=0
MOVL C01151 V=800.0 PL=0
MOVL C01152 V=800.0 PL=0
MOVL C01153 V=800.0 PL=0
MOVL C01154 V=800.0 PL=0
MOVL C01155 V=800.0 PL=0
MOVL C01156 V=800.0 PL=0
MOVL C01157 V=800.0 PL=0
MOVL C01158 V=800.0 PL=0
MOVL C01159 V=800.0 PL=0
MOVL C01160 V=800.0 PL=0
MOVL C01161 V=800.0 PL=0
MOVL C01162 V=800.0 PL=0
MOVL C01163 V=800.0 PL=0
MOVL C01164 V=800.0 PL=0
MOVL C01165 V=800.0 PL=0
MOVL C01166 V=800.0 PL=0
MOVL C01167 V=800.0 PL=0
MOVL C01168 V=800.0 PL=0
MOVL C01169 V=800.0 PL=0
MOVL C01170 V=800.0 PL=0
MOVL C01171 V=800.0 PL=0
MOVL C01172 V=800.0 PL=0
MOVL C01173 V=800.0 PL=0
MOVL C01174 V=800.0 PL=0
MOVL C01175 V=800.0 PL=0
MOVL C01176 V=800.0 PL=0
MOVL C01177 V=800.0 PL=0
MOVL C01178 V=800.0 PL=0
MOVL C01179 V=800.0 PL=0
MOVL C01180 V=800.0 PL=0
MOVL C01181 V=800.0 PL=0
MOVL C01182 V=800.0 PL=0
MOVL C01183 V=800.0 PL=0
MOVL C01184 V=800.0 PL=0
MOVL C01185 V=800.0 PL=0
MOVL C01186 V=800.0 PL=0
MOVL C01187 V=800.0 PL=0
MOVL C01188 V=800.0 PL=0
MOVL C01189 V=800.0 PL=0
MOVL C01190 V=800.0 PL=0
MOVL C01191 V=800.0 PL=0
MOVL C01192 V=800.0 PL=0
MOVL C01193 V=800.0 PL=0
MOVL C01194 V=800.0 PL=0
MOVL C01195 V=800.0 PL=0
MOVL C01196 V=800.0 PL=0
MOVL C01197 V=800.0 PL=0
MOVL C01198 V=800.0 PL=0
MOVL C01199 V=800.0 PL=0
MOVL C01200 V=800.0 PL=0
MOVL C01201 V=800.0 PL=0
MOVL C01202 V=800.0 PL=0
MOVL C01203 V=800.0 PL=0
MOVL C01204 V=800.0 PL=0
MOVL C01205 V=800.0 PL=0
MOVL C01206 V=800.0 PL=0
MOVL C01207 V=800.0 PL=0
MOVL C01208 V=800.0 PL=0
MOVL C01209 V=800.0 PL=0
MOVL C01210 V=800.0 PL=0
MOVL C01211 V=800.0 PL=0
MOVL C01212 V=800.0 PL=0
MOVL C01213 V=800.0 PL=0
MOVL C01214 V=800.0 PL=0
MOVL C01215 V=800.0 PL=0
MOVL C01216 V=800.0 PL=0
MOVL C01217 V=800.0 PL=0
MOVL C01218 V=800.0 PL=0
MOVL C01219 V=800.0 PL=0
MOVL C01220 V=800.0 PL=0
MOVL C01221 V=800.0 PL=0
MOVL C01222 V=800.0 PL=0
MOVL C01223 V=800.0 PL=0
MOVL C01224 V=800.0 PL=0
MOVL C01225 V=800.0 PL=0
MOVL C01226 V=800.0 PL=0
MOVL C01227 V=800.0 PL=0
MOVL C01228 V=800.0 PL=0
MOVL C01229 V=800.0 PL=0
MOVL C01230 V=800.0 PL=0
MOVL C01231 V=800.0 PL=0
MOVL C01232 V=800.0 PL=0
MOVL C01233 V=800.0 PL=0
MOVL C01234 V=800.0 PL=0
MOVL C01235 V=800.0 PL=0
MOVL C01236 V=800.0 PL=0
MOVL C01237 V=800.0 PL=0
MOVL C01238 V=800.0 PL=0
MOVL C01239 V=800.0 PL=0
MOVL C01240 V=800.0 PL=0
MOVL C01241 V=800.0 PL=0
MOVL C01242 V=800.0 PL=0
MOVL C01243 V=800.0 PL=0
MOVL C01244 V=800.0 PL=0
MOVL C01245 V=800.0 PL=0
MOVL C01246 V=800.0 PL=0
MOVL C01247 V=800.0 PL=0
MOVL C01248 V=800.0 PL=0
MOVL C01249 V=800.0 PL=0
MOVL C01250 V=800.0 PL=0
MOVL C01251 V=800.0 PL=0
MOVL C01252 V=800.0 PL=0
MOVL C01253 V=800.0 PL=0
MOVL C01254 V=800.0 PL=0
MOVL C01255 V=800.0 PL=0
MOVL C01256 V=800.0 PL=0
MOVL C01257 V=800.0 PL=0
MOVL C01258 V=800.0 PL=0
MOVL C01259 V=800.0 PL=0
MOVL C01260 V=800.0 PL=0
MOVL C01261 V=800.0 PL=0
MOVL C01262 V=800.0 PL=0
MOVL C01263 V=800.0 PL=0
MOVL C01264 V=800.0 PL=0
MOVL C01265 V=800.0 PL=0
MOVL C01266 V=800.0 PL=0
MOVL C01267 V=800.0 PL=0
MOVL C01268 V=800.0 PL=0
MOVL C01269 V=800.0 PL=0
MOVL C01270 V=800.0 PL=0
MOVL C01271 V=800.0 PL=0
MOVL C01272 V=800.0 PL=0
MOVL C01273 V=800.0 PL=0
MOVL C01274 V=800.0 PL=0
MOVL C01275 V=800.0 PL=0
MOVL C01276 V=800.0 PL=0
MOVL C01277 V=800.0 PL=0
MOVL C01278 V=800.0 PL=0
MOVL C01279 V=800.0 PL=0
MOVL C01280 V=800.0 PL=0
MOVL C01281 V=800.0 PL=0
MOVL C01282 V=800.0 PL=0
MOVL C01283 V=800.0 PL=0
MOVL C01284 V=800.0 PL=0
MOVL C01285 V=800.0 PL=0
MOVL C01286 V=800.0 PL=0
MOVL C01287 V=800.0 PL=0
MOVL C01288 V=800.0 PL=0
MOVL C01289 V=800.0 PL=0
MOVL C01290 V=800.0 PL=0
MOVL C01291 V=800.0 PL=0
MOVL C01292 V=800.0 PL=0
MOVL C01293 V=800.0 PL=0
MOVL C01294 V=800.0 PL=0
MOVL C01295 V=800.0 PL=0
MOVL C01296 V=800.0 PL=0
MOVL C01297 V=800.0 PL=0
MOVL C01298 V=800.0 PL=0
MOVL C01299 V=800.0 PL=0
MOVL C01300 V=800.0 PL=0
MOVL C01301 V=800.0 PL=0
MOVL C01302 V=800.0 PL=0
MOVL C01303 V=800.0 PL=0
MOVL C01304 V=800.0 PL=0
MOVL C01305 V=800.0 PL=0
MOVL C01306 V=800.0 PL=0
MOVL C01307 V=800.0 PL=0
MOVL C01308 V=800.0 PL=0
MOVL C01309 V=800.0 PL=0
MOVL C01310 V=800.0 PL=0
MOVL C01311 V=800.0 PL=0
MOVL C01312 V=800.0 PL=0
MOVL C01313 V=800.0 PL=0
MOVL C01314 V=800.0 PL=0
MOVL C01315 V=800.0 PL=0
MOVL C01316 V=800.0 PL=0
MOVL C01317 V=800.0 PL=0
MOVL C01318 V=800.0 PL=0
MOVL C01319 V=800.0 PL=0
MOVL C01320 V=800.0 PL=0
MOVL C01321 V=800.0 PL=0
MOVL C01322 V=800.0 PL=0
MOVL C01323 V=800.0 PL=0
MOVL C01324 V=800.0 PL=0
MOVL C01325 V=800.0 PL=0
MOVL C01326 V=800.0 PL=0
MOVL C01327 V=800.0 PL=0
MOVL C01328 V=800.0 PL=0
MOVL C01329 V=800.0 PL=0
MOVL C01330 V=800.0 PL=0
MOVL C01331 V=800.0 PL=0
MOVL C01332 V=800.0 PL=0
MOVL C01333 V=800.0 PL=0
MOVL C01334 V=800.0 PL=0
MOVL C01335 V=800.0 PL=0
MOVL C01336 V=800.0 PL=0
MOVL C01337 V=800.0 PL=0
MOVL C01338 V=800.0 PL=0
MOVL C01339 V=800.0 PL=0
MOVL C01340 V=800.0 PL=0
MOVL C01341 V=800.0 PL=0
MOVL C01342 V=800.0 PL=0
MOVL C01343 V=800.0 PL=0
MOVL C01344 V=800.0 PL=0
MOVL C01345 V=800.0 PL=0
MOVL C01346 V=800.0 PL=0
MOVL C01347 V=800.0 PL=0
MOVL C01348 V=800.0 PL=0
MOVL C01349 V=800.0 PL=0
MOVL C01350 V=800.0 PL=0
MOVL C01351 V=800.0 PL=0
MOVL C01352 V=800.0 PL=0
MOVL C01353 V=800.0 PL=0
MOVL C01354 V=800.0 PL=0
MOVL C01355 V=800.0 PL=0
MOVL C01356 V=800.0 PL=0
MOVL C01357 V=800.0 PL=0
MOVL C01358 V=800.0 PL=0
MOVL C01359 V=800.0 PL=0
MOVL C01360 V=800.0 PL=0
MOVL C01361 V=800.0 PL=0
MOVL C01362 V=800.0 PL=0
MOVL C01363 V=800.0 PL=0
MOVL C01364 V=800.0 PL=0
MOVL C01365 V=800.0 PL=0
MOVL C01366 V=800.0 PL=0
MOVL C01367 V=800.0 PL=0
MOVL C01368 V=800.0 PL=0
MOVL C01369 V=800.0 PL=0
MOVL C01370 V=800.0 PL=0
MOVL C01371 V=800.0 PL=0
MOVL C01372 V=800.0 PL=0
MOVL C01373 V=800.0 PL=0
MOVL C01374 V=800.0 PL=0
MOVL C01375 V=800.0 PL=0
MOVL C01376 V=800.0 PL=0
MOVL C01377 V=800.0 PL=0
MOVL C01378 V=800.0 PL=0
MOVL C01379 V=800.0 PL=0
MOVL C01380 V=800.0 PL=0
MOVL C01381 V=800.0 PL=0
MOVL C01382 V=800.0 PL=0
MOVL C01383 V=800.0 PL=0
MOVL C01384 V=800.0 PL=0
MOVL C01385 V=800.0 PL=0
MOVL C01386 V=800.0 PL=0
MOVL C01387 V=800.0 PL=0
MOVL C01388 V=800.0 PL=0
MOVL C01389 V=800.0 PL=0
MOVL C01390 V=800.0 PL=0
MOVL C01391 V=800.0 PL=0
MOVL C01392 V=800.0 PL=0
MOVL C01393 V=800.0 PL=0
MOVL C01394 V=800.0 PL=0
MOVL C01395 V=800.0 PL=0
MOVL C01396 V=800.0 PL=0
MOVL C01397 V=800.0 PL=0
MOVL C01398 V=800.0 PL=0
MOVL C01399 V=800.0 PL=0
MOVL C01400 V=800.0 PL=0
MOVL C01401 V=800.0 PL=0
MOVL C01402 V=800.0 PL=0
MOVL C01403 V=800.0 PL=0
MOVL C01404 V=800.0 PL=0
MOVL C01405 V=800.0 PL=0
MOVL C01406 V=800.0 PL=0
MOVL C01407 V=800.0 PL=0
MOVL C01408 V=800.0 PL=0
MOVL C01409 V=800.0 PL=0
MOVL C01410 V=800.0 PL=0
MOVL C01411 V=800.0 PL=0
MOVL C01412 V=800.0 PL=0
MOVL C01413 V=800.0 PL=0
MOVL C01414 V=800.0 PL=0
MOVL C01415 V=800.0 PL=0
MOVL C01416 V=800.0 PL=0
MOVL C01417 V=800.0 PL=0
MOVL C01418 V=800.0 PL=0
MOVL C01419 V=800.0 PL=0
MOVL C01420 V=800.0 PL=0
MOVL C01421 V=800.0 PL=0
MOVL C01422 V=800.0 PL=0
MOVL C01423 V=800.0 PL=0
MOVL C01424 V=800.0 PL=0
MOVL C01425 V=800.0 PL=0
MOVL C01426 V=800.0 PL=0
MOVL C01427 V=800.0 PL=0
MOVL C01428 V=800.0 PL=0
MOVL C01429 V=800.0 PL=0
MOVL C01430 V=800.0 PL=0
MOVL C01431 V=800.0 PL=0
MOVL C01432 V=800.0 PL=0
MOVL C01433 V=800.0 PL=0
MOVL C01434 V=800.0 PL=0
MOVL C01435 V=800.0 PL=0
MOVL C01436 V=800.0 PL=0
MOVL C01437 V=800.0 PL=0
MOVL C01438 V=800.0 PL=0
MOVL C01439 V=800.0 PL=0
MOVL C01440 V=800.0 PL=0
MOVL C01441 V=800.0 PL=0
MOVL C01442 V=800.0 PL=0
MOVL C01443 V=800.0 PL=0
MOVL C01444 V=800.0 PL=0
MOVL C01445 V=800.0 PL=0
MOVL C01446 V=800.0 PL=0
MOVL C01447 V=800.0 PL=0
MOVL C01448 V=800.0 PL=0
MOVL C01449 V=800.0 PL=0
MOVL C01450 V=800.0 PL=0
MOVL C01451 V=800.0 PL=0
MOVL C01452 V=800.0 PL=0
MOVL C01453 V=800.0 PL=0
MOVL C01454 V=800.0 PL=0
MOVL C01455 V=800.0 PL=0
MOVL C01456 V=800.0 PL=0
MOVL C01457 V=800.0 PL=0
MOVL C01458 V=800.0 PL=0
MOVL C01459 V=800.0 PL=0
MOVL C01460 V=800.0 PL=0
MOVL C01461 V=800.0 PL=0
MOVL C01462 V=800.0 PL=0
MOVL C01463 V=800.0 PL=0
MOVL C01464 V=800.0 PL=0
MOVL C01465 V=800.0 PL=0
MOVL C01466 V=800.0 PL=0
MOVL C01467 V=800.0 PL=0
MOVL C01468 V=800.0 PL=0
MOVL C01469 V=800.0 PL=0
MOVL C01470 V=800.0 PL=0
MOVL C01471 V=800.0 PL=0
MOVL C01472 V=800.0 PL=0
MOVL C01473 V=800.0 PL=0
MOVL C01474 V=800.0 PL=0
MOVL C01475 V=800.0 PL=0
MOVL C01476 V=800.0 PL=0
MOVL C01477 V=800.0 PL=0
MOVL C01478 V=800.0 PL=0
MOVL C01479 V=800.0 PL=0
MOVL C01480 V=800.0 PL=0
MOVL C01481 V=800.0 PL=0
MOVL C01482 V=800.0 PL=0
MOVL C01483 V=800.0 PL=0
MOVL C01484 V=800.0 PL=0
MOVL C01485 V=800.0 PL=0
MOVL C01486 V=800.0 PL=0
MOVL C01487 V=800.0 PL=0
MOVL C01488 V=800.0 PL=0
MOVL C01489 V=800.0 PL=0
MOVL C01490 V=800.0 PL=0
MOVL C01491 V=800.0 PL=0
MOVL C01492 V=800.0 PL=0
MOVL C01493 V=800.0 PL=0
MOVL C01494 V=800.0 PL=0
MOVL C01495 V=800.0 PL=0
MOVL C01496 V=800.0 PL=0
MOVL C01497 V=800.0 PL=0
MOVL C01498 V=800.0 PL=0
MOVL C01499 V=800.0 PL=0
MOVL C01500 V=800.0 PL=0
MOVL C01501 V=800.0 PL=0
MOVL C01502 V=800.0 PL=0
MOVL C01503 V=800.0 PL=0
MOVL C01504 V=800.0 PL=0
MOVL C01505 V=800.0 PL=0
MOVL C01506 V=800.0 PL=0
MOVL C01507 V=800.0 PL=0
MOVL C01508 V=800.0 PL=0
MOVL C01509 V=800.0 PL=0
MOVL C01510 V=800.0 PL=0
MOVL C01511 V=800.0 PL=0
MOVL C01512 V=800.0 PL=0
MOVL C01513 V=800.0 PL=0
MOVL C01514 V=800.0 PL=0
MOVL C01515 V=800.0 PL=0
MOVL C01516 V=800.0 PL=0
MOVL C01517 V=800.0 PL=0
MOVL C01518 V=800.0 PL=0
MOVL C01519 V=800.0 PL=0
MOVL C01520 V=800.0 PL=0
MOVL C01521 V=800.0 PL=0
MOVL C01522 V=800.0 PL=0
MOVL C01523 V=800.0 PL=0
MOVL C01524 V=800.0 PL=0
MOVL C01525 V=800.0 PL=0
MOVL C01526 V=800.0 PL=0
MOVL C01527 V=800.0 PL=0
MOVL C01528 V=800.0 PL=0
MOVL C01529 V=800.0 PL=0
MOVL C01530 V=800.0 PL=0
MOVL C01531 V=800.0 PL=0
MOVL C01532 V=800.0 PL=0
MOVL C01533 V=800.0 PL=0
MOVL C01534 V=800.0 PL=0
MOVL C01535 V=800.0 PL=0
MOVL C01536 V=800.0 PL=0
MOVL C01537 V=800.0 PL=0
MOVL C01538 V=800.0 PL=0
MOVL C01539 V=800.0 PL=0
MOVL C01540 V=800.0 PL=0
MOVL C01541 V=800.0 PL=0
MOVL C01542 V=800.0 PL=0
MOVL C01543 V=800.0 PL=0
MOVL C01544 V=800.0 PL=0
MOVL C01545 V=800.0 PL=0
MOVL C01546 V=800.0 PL=0
MOVL C01547 V=800.0 PL=0
MOVL C01548 V=800.0 PL=0
MOVL C01549 V=800.0 PL=0
MOVL C01550 V=800.0 PL=0
MOVL C01551 V=800.0 PL=0
MOVL C01552 V=800.0 PL=0
MOVL C01553 V=800.0 PL=0
MOVL C01554 V=800.0 PL=0
MOVL C01555 V=800.0 PL=0
MOVL C01556 V=800.0 PL=0
MOVL C01557 V=800.0 PL=0
MOVL C01558 V=800.0 PL=0
MOVL C01559 V=800.0 PL=0
MOVL C01560 V=800.0 PL=0
MOVL C01561 V=800.0 PL=0
MOVL C01562 V=800.0 PL=0
MOVL C01563 V=800.0 PL=0
MOVL C01564 V=800.0 PL=0
MOVL C01565 V=800.0 PL=0
MOVL C01566 V=800.0 PL=0
MOVL C01567 V=800.0 PL=0
MOVL C01568 V=800.0 PL=0
MOVL C01569 V=800.0 PL=0
MOVL C01570 V=800.0 PL=0
MOVL C01571 V=800.0 PL=0
MOVL C01572 V=800.0 PL=0
MOVL C01573 V=800.0 PL=0
MOVL C01574 V=800.0 PL=0
MOVL C01575 V=800.0 PL=0
MOVL C01576 V=800.0 PL=0
MOVL C01577 V=800.0 PL=0
MOVL C01578 V=800.0 PL=0
MOVL C01579 V=800.0 PL=0
MOVL C01580 V=800.0 PL=0
MOVL C01581 V=800.0 PL=0
MOVL C01582 V=800.0 PL=0
MOVL C01583 V=800.0 PL=0
MOVL C01584 V=800.0 PL=0
MOVL C01585 V=800.0 PL=0
MOVL C01586 V=800.0 PL=0
MOVL C01587 V=800.0 PL=0
MOVL C01588 V=800.0 PL=0
MOVL C01589 V=800.0 PL=0
MOVL C01590 V=800.0 PL=0
MOVL C01591 V=800.0 PL=0
MOVL C01592 V=800.0 PL=0
MOVL C01593 V=800.0 PL=0
MOVL C01594 V=800.0 PL=0
MOVL C01595 V=800.0 PL=0
MOVL C01596 V=800.0 PL=0
MOVL C01597 V=800.0 PL=0
MOVL C01598 V=800.0 PL=0
MOVL C01599 V=800.0 PL=0
MOVL C01600 V=800.0 PL=0
MOVL C01601 V=800.0 PL=0
MOVL C01602 V=800.0 PL=0
MOVL C01603 V=800.0 PL=0
MOVL C01604 V=800.0 PL=0
MOVL C01605 V=800.0 PL=0
MOVL C01606 V=800.0 PL=0
MOVL C01607 V=800.0 PL=0
MOVL C01608 V=800.0 PL=0
MOVL C01609 V=800.0 PL=0
MOVL C01610 V=800.0 PL=0
MOVL C01611 V=800.0 PL=0
MOVL C01612 V=800.0 PL=0
MOVL C01613 V=800.0 PL=0
MOVL C01614 V=800.0 PL=0
MOVL C01615 V=800.0 PL=0
MOVL C01616 V=800.0 PL=0
MOVL C01617 V=800.0 PL=0
MOVL C01618 V=800.0 PL=0
MOVL C01619 V=800.0 PL=0
MOVL C01620 V=800.0 PL=0
MOVL C01621 V=800.0 PL=0
MOVL C01622 V=800.0 PL=0
MOVL C01623 V=800.0 PL=0
MOVL C01624 V=800.0 PL=0
MOVL C01625 V=800.0 PL=0
MOVL C01626 V=800.0 PL=0
MOVL C01627 V=800.0 PL=0
MOVL C01628 V=800.0 PL=0
MOVL C01629 V=800.0 PL=0
MOVL C01630 V=800.0 PL=0
MOVL C01631 V=800.0 PL=0
MOVL C01632 V=800.0 PL=0
MOVL C01633 V=800.0 PL=0
MOVL C01634 V=800.0 PL=0
MOVL C01635 V=800.0 PL=0
MOVL C01636 V=800.0 PL=0
MOVL C01637 V=800.0 PL=0
MOVL C01638 V=800.0 PL=0
MOVL C01639 V=800.0 PL=0
MOVL C01640 V=800.0 PL=0
MOVL C01641 V=800.0 PL=0
MOVL C01642 V=800.0 PL=0
MOVL C01643 V=800.0 PL=0
MOVL C01644 V=800.0 PL=0
MOVL C01645 V=800.0 PL=0
MOVL C01646 V=800.0 PL=0
MOVL C01647 V=800.0 PL=0
MOVL C01648 V=800.0 PL=0
MOVL C01649 V=800.0 PL=0
MOVL C01650 V=800.0 PL=0
MOVL C01651 V=800.0 PL=0
MOVL C01652 V=800.0 PL=0
MOVL C01653 V=800.0 PL=0
MOVL C01654 V=800.0 PL=0
MOVL C01655 V=800.0 PL=0
MOVL C01656 V=800.0 PL=0
MOVL C01657 V=800.0 PL=0
MOVL C01658 V=800.0 PL=0
MOVL C01659 V=800.0 PL=0
MOVL C01660 V=800.0 PL=0
MOVL C01661 V=800.0 PL=0
MOVL C01662 V=800.0 PL=0
MOVL C01663 V=800.0 PL=0
MOVL C01664 V=800.0 PL=0
MOVL C01665 V=800.0 PL=0
MOVL C01666 V=800.0 PL=0
MOVL C01667 V=800.0 PL=0
MOVL C01668 V=800.0 PL=0
MOVL C01669 V=800.0 PL=0
MOVL C01670 V=800.0 PL=0
MOVL C01671 V=800.0 PL=0
MOVL C01672 V=800.0 PL=0
MOVL C01673 V=800.0 PL=0
MOVL C01674 V=800.0 PL=0
MOVL C01675 V=800.0 PL=0
MOVL C01676 V=800.0 PL=0
MOVL C01677 V=800.0 PL=0
MOVL C01678 V=800.0 PL=0
MOVL C01679 V=800.0 PL=0
MOVL C01680 V=800.0 PL=0
MOVL C01681 V=800.0 PL=0
MOVL C01682 V=800.0 PL=0
MOVL C01683 V=800.0 PL=0
MOVL C01684 V=800.0 PL=0
MOVL C01685 V=800.0 PL=0
MOVL C01686 V=800.0 PL=0
MOVL C01687 V=800.0 PL=0
MOVL C01688 V=800.0 PL=0
MOVL C01689 V=800.0 PL=0
MOVL C01690 V=800.0 PL=0
MOVL C01691 V=800.0 PL=0
MOVL C01692 V=800.0 PL=0
MOVL C01693 V=800.0 PL=0
MOVL C01694 V=800.0 PL=0
MOVL C01695 V=800.0 PL=0
MOVL C01696 V=800.0 PL=0
MOVL C01697 V=800.0 PL=0
MOVL C01698 V=800.0 PL=0
MOVL C01699 V=800.0 PL=0
MOVL C01700 V=800.0 PL=0
MOVL C01701 V=800.0 PL=0
MOVL C01702 V=800.0 PL=0
MOVL C01703 V=800.0 PL=0
MOVL C01704 V=800.0 PL=0
MOVL C01705 V=800.0 PL=0
MOVL C01706 V=800.0 PL=0
MOVL C01707 V=800.0 PL=0
MOVL C01708 V=800.0 PL=0
MOVL C01709 V=800.0 PL=0
MOVL C01710 V=800.0 PL=0
MOVL C01711 V=800.0 PL=0
MOVL C01712 V=800.0 PL=0
MOVL C01713 V=800.0 PL=0
MOVL C01714 V=800.0 PL=0
MOVL C01715 V=800.0 PL=0
MOVL C01716 V=800.0 PL=0
MOVL C01717 V=800.0 PL=0
MOVL C01718 V=800.0 PL=0
MOVL C01719 V=800.0 PL=0
MOVL C01720 V=800.0 PL=0
MOVL C01721 V=800.0 PL=0
MOVL C01722 V=800.0 PL=0
MOVL C01723 V=800.0 PL=0
MOVL C01724 V=800.0 PL=0
MOVL C01725 V=800.0 PL=0
MOVL C01726 V=800.0 PL=0
MOVL C01727 V=800.0 PL=0
MOVL C01728 V=800.0 PL=0
MOVL C01729 V=800.0 PL=0
MOVL C01730 V=800.0 PL=0
MOVL C01731 V=800.0 PL=0
MOVL C01732 V=800.0 PL=0
MOVL C01733 V=800.0 PL=0
MOVL C01734 V=800.0 PL=0
MOVL C01735 V=800.0 PL=0
MOVL C01736 V=800.0 PL=0
MOVL C01737 V=800.0 PL=0
MOVL C01738 V=800.0 PL=0
MOVL C01739 V=800.0 PL=0
MOVL C01740 V=800.0 PL=0
MOVL C01741 V=800.0 PL=0
MOVL C01742 V=800.0 PL=0
MOVL C01743 V=800.0 PL=0
MOVL C01744 V=800.0 PL=0
MOVL C01745 V=800.0 PL=0
MOVL C01746 V=800.0 PL=0
MOVL C01747 V=800.0 PL=0
MOVL C01748 V=800.0 PL=0
MOVL C01749 V=800.0 PL=0
MOVL C01750 V=800.0 PL=0
MOVL C01751 V=800.0 PL=0
MOVL C01752 V=800.0 PL=0
MOVL C01753 V=800.0 PL=0
MOVL C01754 V=800.0 PL=0
MOVL C01755 V=800.0 PL=0
MOVL C01756 V=800.0 PL=0
MOVL C01757 V=800.0 PL=0
MOVL C01758 V=800.0 PL=0
MOVL C01759 V=800.0 PL=0
MOVL C01760 V=800.0 PL=0
MOVL C01761 V=800.0 PL=0
MOVL C01762 V=800.0 PL=0
MOVL C01763 V=800.0 PL=0
MOVL C01764 V=800.0 PL=0
MOVL C01765 V=800.0 PL=0
MOVL C01766 V=800.0 PL=0
MOVL C01767 V=800.0 PL=0
MOVL C01768 V=800.0 PL=0
MOVL C01769 V=800.0 PL=0
MOVL C01770 V=800.0 PL=0
MOVL C01771 V=800.0 PL=0
MOVL C01772 V=800.0 PL=0
MOVL C01773 V=800.0 PL=0
MOVL C01774 V=800.0 PL=0
MOVL C01775 V=800.0 PL=0
MOVL C01776 V=800.0 PL=0
MOVL C01777 V=800.0 PL=0
MOVL C01778 V=800.0 PL=0
MOVL C01779 V=800.0 PL=0
MOVL C01780 V=800.0 PL=0
MOVL C01781 V=800.0 PL=0
MOVL C01782 V=800.0 PL=0
MOVL C01783 V=800.0 PL=0
MOVL C01784 V=800.0 PL=0
MOVL C01785 V=800.0 PL=0
MOVL C01786 V=800.0 PL=0
MOVL C01787 V=800.0 PL=0
MOVL C01788 V=800.0 PL=0
MOVL C01789 V=800.0 PL=0
MOVL C01790 V=800.0 PL=0
MOVL C01791 V=800.0 PL=0
MOVL C01792 V=800.0 PL=0
MOVL C01793 V=800.0 PL=0
MOVL C01794 V=800.0 PL=0
MOVL C01795 V=800.0 PL=0
MOVL C01796 V=800.0 PL=0
MOVL C01797 V=800.0 PL=0
MOVL C01798 V=800.0 PL=0
MOVL C01799 V=800.0 PL=0
MOVL C01800 V=800.0 PL=0
MOVL C01801 V=800.0 PL=0
MOVL C01802 V=800.0 PL=0
MOVL C01803 V=800.0 PL=0
MOVL C01804 V=800.0 PL=0
MOVL C01805 V=800.0 PL=0
MOVL C01806 V=800.0 PL=0
MOVL C01807 V=800.0 PL=0
MOVL C01808 V=800.0 PL=0
MOVL C01809 V=800.0 PL=0
MOVL C01810 V=800.0 PL=0
MOVL C01811 V=800.0 PL=0
MOVL C01812 V=800.0 PL=0
MOVL C01813 V=800.0 PL=0
MOVL C01814 V=800.0 PL=0
MOVL C01815 V=800.0 PL=0
MOVL C01816 V=800.0 PL=0
MOVL C01817 V=800.0 PL=0
MOVL C01818 V=800.0 PL=0
MOVL C01819 V=800.0 PL=0
MOVL C01820 V=800.0 PL=0
MOVL C01821 V=800.0 PL=0
MOVL C01822 V=800.0 PL=0
MOVL C01823 V=800.0 PL=0
MOVL C01824 V=800.0 PL=0
MOVL C01825 V=800.0 PL=0
MOVL C01826 V=800.0 PL=0
MOVL C01827 V=800.0 PL=0
MOVL C01828 V=800.0 PL=0
MOVL C01829 V=800.0 PL=0
MOVL C01830 V=800.0 PL=0
MOVL C01831 V=800.0 PL=0
MOVL C01832 V=800.0 PL=0
MOVL C01833 V=800.0 PL=0
MOVL C01834 V=800.0 PL=0
MOVL C01835 V=800.0 PL=0
MOVL C01836 V=800.0 PL=0
MOVL C01837 V=800.0 PL=0
MOVL C01838 V=800.0 PL=0
MOVL C01839 V=800.0 PL=0
MOVL C01840 V=800.0 PL=0
MOVL C01841 V=800.0 PL=0
MOVL C01842 V=800.0 PL=0
MOVL C01843 V=800.0 PL=0
MOVL C01844 V=800.0 PL=0
MOVL C01845 V=800.0 PL=0
MOVL C01846 V=800.0 PL=0
MOVL C01847 V=800.0 PL=0
MOVL C01848 V=800.0 PL=0
MOVL C01849 V=800.0 PL=0
MOVL C01850 V=800.0 PL=0
MOVL C01851 V=800.0 PL=0
MOVL C01852 V=800.0 PL=0
MOVL C01853 V=800.0 PL=0
MOVL C01854 V=800.0 PL=0
MOVL C01855 V=800.0 PL=0
MOVL C01856 V=800.0 PL=0
MOVL C01857 V=800.0 PL=0
MOVL C01858 V=800.0 PL=0
MOVL C01859 V=800.0 PL=0
MOVL C01860 V=800.0 PL=0
MOVL C01861 V=800.0 PL=0
MOVL C01862 V=800.0 PL=0
MOVL C01863 V=800.0 PL=0
MOVL C01864 V=800.0 PL=0
MOVL C01865 V=800.0 PL=0
MOVL C01866 V=800.0 PL=0
MOVL C01867 V=800.0 PL=0
MOVL C01868 V=800.0 PL=0
MOVL C01869 V=800.0 PL=0
MOVL C01870 V=800.0 PL=0
MOVL C01871 V=800.0 PL=0
MOVL C01872 V=800.0 PL=0
MOVL C01873 V=800.0 PL=0
MOVL C01874 V=800.0 PL=0
MOVL C01875 V=800.0 PL=0
MOVL C01876 V=800.0 PL=0
MOVL C01877 V=800.0 PL=0
MOVL C01878 V=800.0 PL=0
MOVL C01879 V=800.0 PL=0
MOVL C01880 V=800.0 PL=0
MOVL C01881 V=800.0 PL=0
MOVL C01882 V=800.0 PL=0
MOVL C01883 V=800.0 PL=0
MOVL C01884 V=800.0 PL=0
MOVL C01885 V=800.0 PL=0
MOVL C01886 V=800.0 PL=0
MOVL C01887 V=800.0 PL=0
MOVL C01888 V=800.0 PL=0
MOVL C01889 V=800.0 PL=0
MOVL C01890 V=800.0 PL=0
MOVL C01891 V=800.0 PL=0
MOVL C01892 V=800.0 PL=0
MOVL C01893 V=800.0 PL=0
MOVL C01894 V=800.0 PL=0
MOVL C01895 V=800.0 PL=0
MOVL C01896 V=800.0 PL=0
MOVL C01897 V=800.0 PL=0
MOVL C01898 V=800.0 PL=0
MOVL C01899 V=800.0 PL=0
MOVL C01900 V=800.0 PL=0
MOVL C01901 V=800.0 PL=0
MOVL C01902 V=800.0 PL=0
MOVL C01903 V=800.0 PL=0
MOVL C01904 V=800.0 PL=0
MOVL C01905 V=800.0 PL=0
MOVL C01906 V=800.0 PL=0
MOVL C01907 V=800.0 PL=0
MOVL C01908 V=800.0 PL=0
MOVL C01909 V=800.0 PL=0
MOVL C01910 V=800.0 PL=0
MOVL C01911 V=800.0 PL=0
MOVL C01912 V=800.0 PL=0
MOVL C01913 V=800.0 PL=0
MOVL C01914 V=800.0 PL=0
MOVL C01915 V=800.0 PL=0
MOVL C01916 V=800.0 PL=0
MOVL C01917 V=800.0 PL=0
MOVL C01918 V=800.0 PL=0
MOVL C01919 V=800.0 PL=0
MOVL C01920 V=800.0 PL=0
MOVL C01921 V=800.0 PL=0
MOVL C01922 V=800.0 PL=0
MOVL C01923 V=800.0 PL=0
MOVL C01924 V=800.0 PL=0
MOVL C01925 V=800.0 PL=0
MOVL C01926 V=800.0 PL=0
MOVL C01927 V=800.0 PL=0
MOVL C01928 V=800.0 PL=0
MOVL C01929 V=800.0 PL=0
MOVL C01930 V=800.0 PL=0
MOVL C01931 V=800.0 PL=0
MOVL C01932 V=800.0 PL=0
MOVL C01933 V=800.0 PL=0
MOVL C01934 V=800.0 PL=0
MOVL C01935 V=800.0 PL=0
MOVL C01936 V=800.0 PL=0
MOVL C01937 V=800.0 PL=0
MOVL C01938 V=800.0 PL=0
MOVL C01939 V=800.0 PL=0
MOVL C01940 V=800.0 PL=0
MOVL C01941 V=800.0 PL=0
MOVL C01942 V=800.0 PL=0
MOVL C01943 V=800.0 PL=0
MOVL C01944 V=800.0 PL=0
MOVL C01945 V=800.0 PL=0
MOVL C01946 V=800.0 PL=0
MOVL C01947 V=800.0 PL=0
MOVL C01948 V=800.0 PL=0
MOVL C01949 V=800.0 PL=0
MOVL C01950 V=800.0 PL=0
MOVL C01951 V=800.0 PL=0
MOVL C01952 V=800.0 PL=0
MOVL C01953 V=800.0 PL=0
MOVL C01954 V=800.0 PL=0
MOVL C01955 V=800.0 PL=0
MOVL C01956 V=800.0 PL=0
MOVL C01957 V=800.0 PL=0
MOVL C01958 V=800.0 PL=0
MOVL C01959 V=800.0 PL=0
MOVL C01960 V=800.0 PL=0
MOVL C01961 V=800.0 PL=0
MOVL C01962 V=800.0 PL=0
MOVL C01963 V=800.0 PL=0
MOVL C01964 V=800.0 PL=0
MOVL C01965 V=800.0 PL=0
MOVL C01966 V=800.0 PL=0
MOVL C01967 V=800.0 PL=0
MOVL C01968 V=800.0 PL=0
MOVL C01969 V=800.0 PL=0
MOVL C01970 V=800.0 PL=0
MOVL C01971 V=800.0 PL=0
MOVL C01972 V=800.0 PL=0
MOVL C01973 V=800.0 PL=0
MOVL C01974 V=800.0 PL=0
MOVL C01975 V=800.0 PL=0
MOVL C01976 V=800.0 PL=0
MOVL C01977 V=800.0 PL=0
MOVL C01978 V=800.0 PL=0
MOVL C01979 V=800.0 PL=0
MOVL C01980 V=800.0 PL=0
MOVL C01981 V=800.0 PL=0
MOVL C01982 V=800.0 PL=0
MOVL C01983 V=800.0 PL=0
MOVL C01984 V=800.0 PL=0
MOVL C01985 V=800.0 PL=0
MOVL C01986 V=800.0 PL=0
MOVL C01987 V=800.0 PL=0
MOVL C01988 V=800.0 PL=0
MOVL C01989 V=800.0 PL=0
MOVL C01990 V=800.0 PL=0
MOVL C01991 V=800.0 PL=0
MOVL C01992 V=800.0 PL=0
MOVL C01993 V=800.0 PL=0
MOVL C01994 V=800.0 PL=0
MOVL C01995 V=800.0 PL=0
MOVL C01996 V=800.0 PL=0
MOVL C01997 V=800.0 PL=0
MOVL C01998 V=800.0 PL=0
MOVL C01999 V=800.0 PL=0
MOVL C02000 V=800.0 PL=0
MOVL C02001 V=800.0 PL=0
MOVL C02002 V=800.0 PL=0
MOVL C02003 V=800.0 PL=0
MOVL C02004 V=800.0 PL=0
MOVL C02005 V=800.0 PL=0
MOVL C02006 V=800.0 PL=0
MOVL C02007 V=800.0 PL=0
MOVL C02008 V=800.0 PL=0
MOVL C02009 V=800.0 PL=0
MOVL C02010 V=800.0 PL=0
MOVL C02011 V=800.0 PL=0
MOVL C02012 V=800.0 PL=0
MOVL C02013 V=800.0 PL=0
MOVL C02014 V=800.0 PL=0
MOVL C02015 V=800.0 PL=0
MOVL C02016 V=800.0 PL=0
MOVL C02017 V=800.0 PL=0
MOVL C02018 V=800.0 PL=0
MOVL C02019 V=800.0 PL=0
MOVL C02020 V=800.0 PL=0
MOVL C02021 V=800.0 PL=0
MOVL C02022 V=800.0 PL=0
MOVL C02023 V=800.0 PL=0
MOVL C02024 V=800.0 PL=0
MOVL C02025 V=800.0 PL=0
MOVL C02026 V=800.0 PL=0
MOVL C02027 V=800.0 PL=0
MOVL C02028 V=800.0 PL=0
MOVL C02029 V=800.0 PL=0
MOVL C02030 V=800.0 PL=0
MOVL C02031 V=800.0 PL=0
MOVL C02032 V=800.0 PL=0
MOVL C02033 V=800.0 PL=0
MOVL C02034 V=800.0 PL=0
MOVL C02035 V=800.0 PL=0
MOVL C02036 V=800.0 PL=0
MOVL C02037 V=800.0 PL=0
MOVL C02038 V=800.0 PL=0
MOVL C02039 V=800.0 PL=0
MOVL C02040 V=800.0 PL=0
MOVL C02041 V=800.0 PL=0
MOVL C02042 V=800.0 PL=0
MOVL C02043 V=800.0 PL=0
MOVL C02044 V=800.0 PL=0
MOVL C02045 V=800.0 PL=0
MOVL C02046 V=800.0 PL=0
MOVL C02047 V=800.0 PL=0
MOVL C02048 V=800.0 PL=0
MOVL C02049 V=800.0 PL=0
MOVL C02050 V=800.0 PL=0
MOVL C02051 V=800.0 PL=0
MOVL C02052 V=800.0 PL=0
MOVL C02053 V=800.0 PL=0
MOVL C02054 V=800.0 PL=0
MOVL C02055 V=800.0 PL=0
MOVL C02056 V=800.0 PL=0
MOVL C02057 V=800.0 PL=0
MOVL C02058 V=800.0 PL=0
MOVL C02059 V=800.0 PL=0
MOVL C02060 V=800.0 PL=0
MOVL C02061 V=800.0 PL=0
MOVL C02062 V=800.0 PL=0
MOVL C02063 V=800.0 PL=0
MOVL C02064 V=800.0 PL=0
MOVL C02065 V=800.0 PL=0
MOVL C02066 V=800.0 PL=0
MOVL C02067 V=800.0 PL=0
MOVL C02068 V=800.0 PL=0
MOVL C02069 V=800.0 PL=0
MOVL C02070 V=800.0 PL=0
MOVL C02071 V=800.0 PL=0
MOVL C02072 V=800.0 PL=0
MOVL C02073 V=800.0 PL=0
MOVL C02074 V=800.0 PL=0
MOVL C02075 V=800.0 PL=0
MOVL C02076 V=800.0 PL=0
MOVL C02077 V=800.0 PL=0
MOVL C02078 V=800.0 PL=0
MOVL C02079 V=800.0 PL=0
MOVL C02080 V=800.0 PL=0
MOVL C02081 V=800.0 PL=0
MOVL C02082 V=800.0 PL=0
MOVL C02083 V=800.0 PL=0
MOVL C02084 V=800.0 PL=0
MOVL C02085 V=800.0 PL=0
MOVL C02086 V=800.0 PL=0
MOVL C02087 V=800.0 PL=0
MOVL C02088 V=800.0 PL=0
MOVL C02089 V=800.0 PL=0
MOVL C02090 V=800.0 PL=0
MOVL C02091 V=800.0 PL=0
MOVL C02092 V=800.0 PL=0
MOVL C02093 V=800.0 PL=0
MOVL C02094 V=800.0 PL=0
MOVL C02095 V=800.0 PL=0
MOVL C02096 V=800.0 PL=0
MOVL C02097 V=800.0 PL=0
